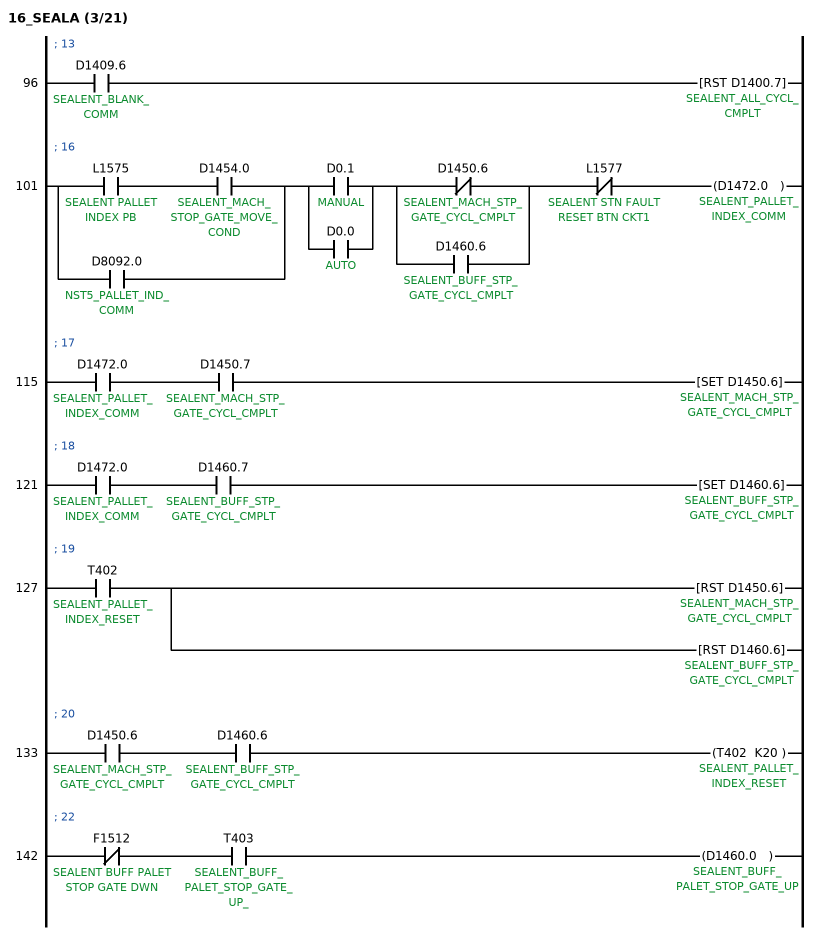
[picture p288: ladder of 16_SEALA, rungs at steps 96 to 142]
; 13
96    LD      D1409.6  ; SEALENT_BLANK_COMM
      RST     D1400.7  ; SEALENT_ALL_CYCL_CMPLT
; 16
101   LD      L1575  ; SEALENT PALLET INDEX PB
      AND     D1454.0  ; SEALENT_MACH_STOP_GATE_MOVE_COND
      OR      D8092.0  ; NST5_PALLET_IND_COMM
      LD      D0.1  ; MANUAL
      OR      D0.0  ; AUTO
      ANB
      LDI     D1450.6  ; SEALENT_MACH_STP_GATE_CYCL_CMPLT
      OR      D1460.6  ; SEALENT_BUFF_STP_GATE_CYCL_CMPLT
      ANB
      ANI     L1577  ; SEALENT STN FAULT RESET BTN CKT1
      OUT     D1472.0  ; SEALENT_PALLET_INDEX_COMM
; 17
115   LD      D1472.0  ; SEALENT_PALLET_INDEX_COMM
      AND     D1450.7  ; SEALENT_MACH_STP_GATE_CYCL_CMPLT
      SET     D1450.6  ; SEALENT_MACH_STP_GATE_CYCL_CMPLT
; 18
121   LD      D1472.0  ; SEALENT_PALLET_INDEX_COMM
      AND     D1460.7  ; SEALENT_BUFF_STP_GATE_CYCL_CMPLT
      SET     D1460.6  ; SEALENT_BUFF_STP_GATE_CYCL_CMPLT
; 19
127   LD      T402  ; SEALENT_PALLET_INDEX_RESET
      RST     D1450.6  ; SEALENT_MACH_STP_GATE_CYCL_CMPLT
      RST     D1460.6  ; SEALENT_BUFF_STP_GATE_CYCL_CMPLT
; 20
133   LD      D1450.6  ; SEALENT_MACH_STP_GATE_CYCL_CMPLT
      AND     D1460.6  ; SEALENT_BUFF_STP_GATE_CYCL_CMPLT
      OUT     T402 K20  ; SEALENT_PALLET_INDEX_RESET
; 22
142   LDI     F1512  ; SEALENT BUFF PALET STOP GATE DWN
      AND     T403  ; SEALENT_BUFF_PALET_STOP_GATE_UP_
      OUT     D1460.0  ; SEALENT_BUFF_PALET_STOP_GATE_UP
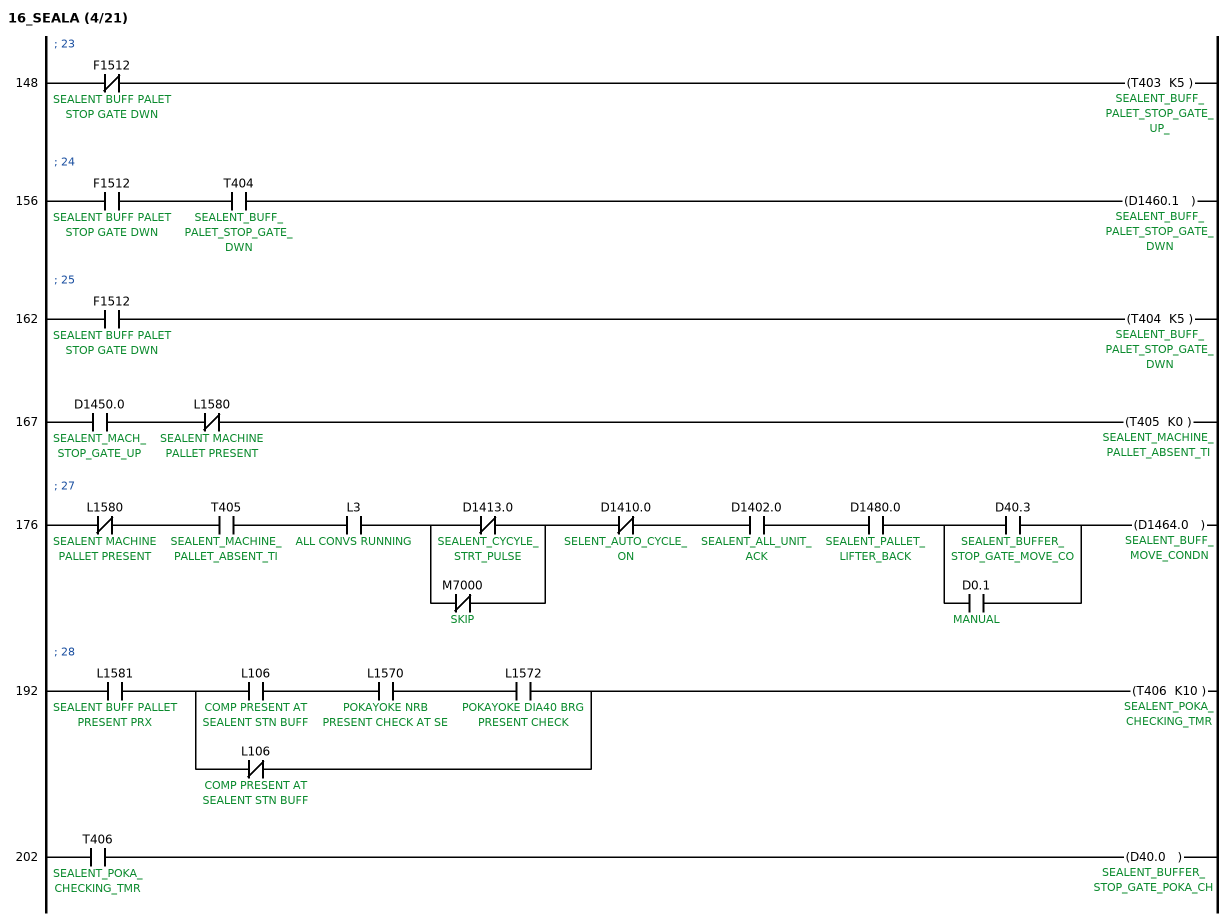
; 23
148   LDI     F1512  ; SEALENT BUFF PALET STOP GATE DWN
      OUT     T403 K5  ; SEALENT_BUFF_PALET_STOP_GATE_UP_
; 24
156   LD      F1512  ; SEALENT BUFF PALET STOP GATE DWN
      AND     T404  ; SEALENT_BUFF_PALET_STOP_GATE_DWN
      OUT     D1460.1  ; SEALENT_BUFF_PALET_STOP_GATE_DWN
; 25
162   LD      F1512  ; SEALENT BUFF PALET STOP GATE DWN
      OUT     T404 K5  ; SEALENT_BUFF_PALET_STOP_GATE_DWN
167   LD      D1450.0  ; SEALENT_MACH_STOP_GATE_UP
      ANI     L1580  ; SEALENT MACHINE PALLET PRESENT
      OUT     T405 K0  ; SEALENT_MACHINE_PALLET_ABSENT_TI
; 27
176   LDI     L1580  ; SEALENT MACHINE PALLET PRESENT
      AND     T405  ; SEALENT_MACHINE_PALLET_ABSENT_TI
      AND     L3  ; ALL CONVS RUNNING
      LDI     D1413.0  ; SEALENT_CYCYLE_STRT_PULSE
      ORI     M7000  ; SKIP
      ANB
      ANI     D1410.0  ; SELENT_AUTO_CYCLE_ON
      AND     D1402.0  ; SEALENT_ALL_UNIT_ACK
      AND     D1480.0  ; SEALENT_PALLET_LIFTER_BACK
      LD      D40.3  ; SEALENT_BUFFER_STOP_GATE_MOVE_CO
      OR      D0.1  ; MANUAL
      ANB
      OUT     D1464.0  ; SEALENT_BUFF_MOVE_CONDN
; 28
192   LD      L1581  ; SEALENT BUFF PALLET PRESENT PRX
      LD      L106  ; COMP PRESENT AT SEALENT STN BUFF
      AND     L1570  ; POKAYOKE NRB PRESENT CHECK AT SE
      AND     L1572  ; POKAYOKE DIA40 BRG PRESENT CHECK
      ORI     L106  ; COMP PRESENT AT SEALENT STN BUFF
      ANB
      OUT     T406 K10  ; SEALENT_POKA_CHECKING_TMR
202   LD      T406  ; SEALENT_POKA_CHECKING_TMR
      OUT     D40.0  ; SEALENT_BUFFER_STOP_GATE_POKA_CH
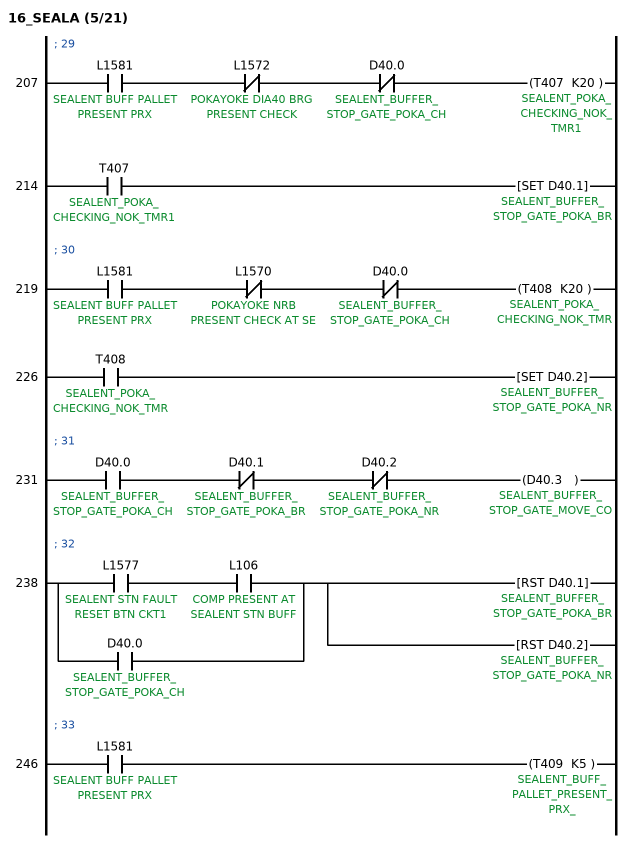
; 29
207   LD      L1581  ; SEALENT BUFF PALLET PRESENT PRX
      ANI     L1572  ; POKAYOKE DIA40 BRG PRESENT CHECK
      ANI     D40.0  ; SEALENT_BUFFER_STOP_GATE_POKA_CH
      OUT     T407 K20  ; SEALENT_POKA_CHECKING_NOK_TMR1
214   LD      T407  ; SEALENT_POKA_CHECKING_NOK_TMR1
      SET     D40.1  ; SEALENT_BUFFER_STOP_GATE_POKA_BR
; 30
219   LD      L1581  ; SEALENT BUFF PALLET PRESENT PRX
      ANI     L1570  ; POKAYOKE NRB PRESENT CHECK AT SE
      ANI     D40.0  ; SEALENT_BUFFER_STOP_GATE_POKA_CH
      OUT     T408 K20  ; SEALENT_POKA_CHECKING_NOK_TMR
226   LD      T408  ; SEALENT_POKA_CHECKING_NOK_TMR
      SET     D40.2  ; SEALENT_BUFFER_STOP_GATE_POKA_NR
; 31
231   LD      D40.0  ; SEALENT_BUFFER_STOP_GATE_POKA_CH
      ANI     D40.1  ; SEALENT_BUFFER_STOP_GATE_POKA_BR
      ANI     D40.2  ; SEALENT_BUFFER_STOP_GATE_POKA_NR
      OUT     D40.3  ; SEALENT_BUFFER_STOP_GATE_MOVE_CO
; 32
238   LD      L1577  ; SEALENT STN FAULT RESET BTN CKT1
      AND     L106  ; COMP PRESENT AT SEALENT STN BUFF
      OR      D40.0  ; SEALENT_BUFFER_STOP_GATE_POKA_CH
      RST     D40.1  ; SEALENT_BUFFER_STOP_GATE_POKA_BR
      RST     D40.2  ; SEALENT_BUFFER_STOP_GATE_POKA_NR
; 33
246   LD      L1581  ; SEALENT BUFF PALLET PRESENT PRX
      OUT     T409 K5  ; SEALENT_BUFF_PALLET_PRESENT_PRX_
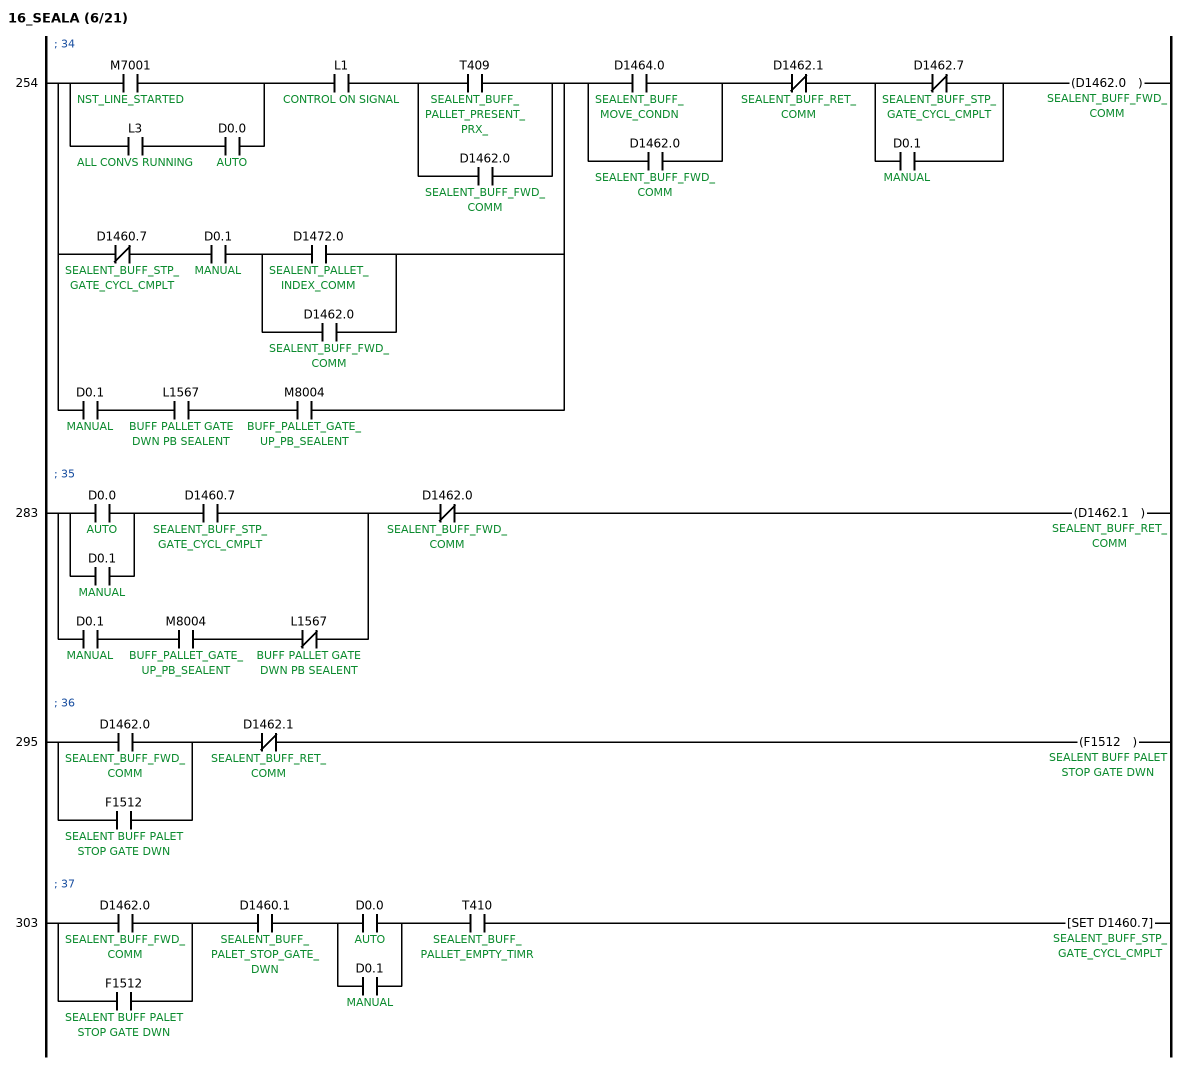
; 34
254   LD      M7001  ; NST_LINE_STARTED
      LD      L3  ; ALL CONVS RUNNING
      AND     D0.0  ; AUTO
      ORB
      AND     L1  ; CONTROL ON SIGNAL
      LD      T409  ; SEALENT_BUFF_PALLET_PRESENT_PRX_
      OR      D1462.0  ; SEALENT_BUFF_FWD_COMM
      ANB
      LDI     D1460.7  ; SEALENT_BUFF_STP_GATE_CYCL_CMPLT
      AND     D0.1  ; MANUAL
      LD      D1472.0  ; SEALENT_PALLET_INDEX_COMM
      OR      D1462.0  ; SEALENT_BUFF_FWD_COMM
      ANB
      ORB
      LD      D0.1  ; MANUAL
      AND     L1567  ; BUFF PALLET GATE DWN PB SEALENT
      AND     M8004  ; BUFF_PALLET_GATE_UP_PB_SEALENT
      ORB
      LD      D1464.0  ; SEALENT_BUFF_MOVE_CONDN
      OR      D1462.0  ; SEALENT_BUFF_FWD_COMM
      ANB
      ANI     D1462.1  ; SEALENT_BUFF_RET_COMM
      LDI     D1462.7  ; SEALENT_BUFF_STP_GATE_CYCL_CMPLT
      OR      D0.1  ; MANUAL
      ANB
      OUT     D1462.0  ; SEALENT_BUFF_FWD_COMM
; 35
283   LD      D0.0  ; AUTO
      OR      D0.1  ; MANUAL
      AND     D1460.7  ; SEALENT_BUFF_STP_GATE_CYCL_CMPLT
      LD      D0.1  ; MANUAL
      AND     M8004  ; BUFF_PALLET_GATE_UP_PB_SEALENT
      ANI     L1567  ; BUFF PALLET GATE DWN PB SEALENT
      ORB
      ANI     D1462.0  ; SEALENT_BUFF_FWD_COMM
      OUT     D1462.1  ; SEALENT_BUFF_RET_COMM
; 36
295   LD      D1462.0  ; SEALENT_BUFF_FWD_COMM
      OR      F1512  ; SEALENT BUFF PALET STOP GATE DWN
      ANI     D1462.1  ; SEALENT_BUFF_RET_COMM
      OUT     F1512  ; SEALENT BUFF PALET STOP GATE DWN
; 37
303   LD      D1462.0  ; SEALENT_BUFF_FWD_COMM
      OR      F1512  ; SEALENT BUFF PALET STOP GATE DWN
      AND     D1460.1  ; SEALENT_BUFF_PALET_STOP_GATE_DWN
      LD      D0.0  ; AUTO
      OR      D0.1  ; MANUAL
      ANB
      AND     T410  ; SEALENT_BUFF_PALLET_EMPTY_TIMR
      SET     D1460.7  ; SEALENT_BUFF_STP_GATE_CYCL_CMPLT
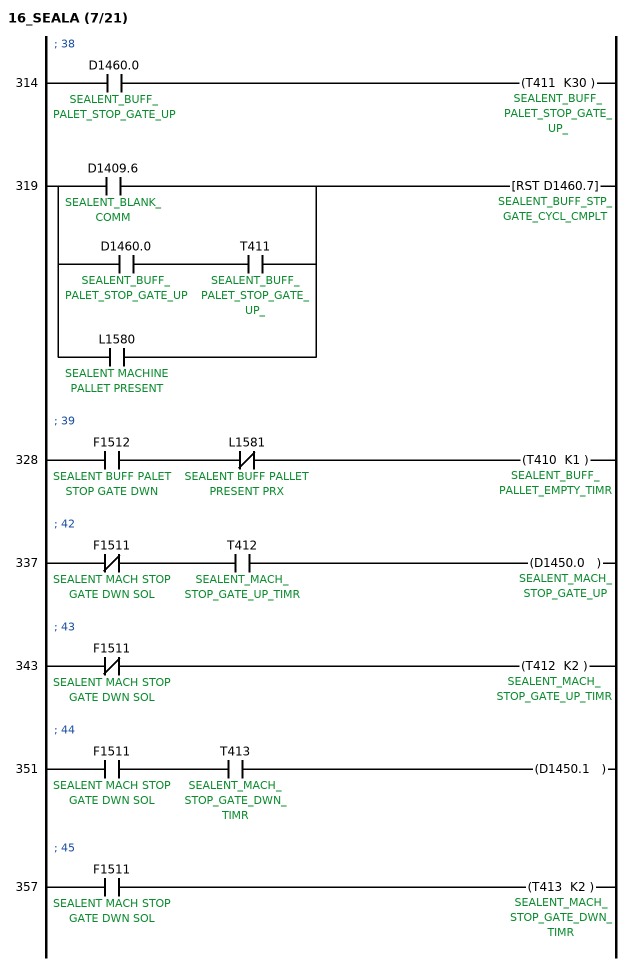
; 38
314   LD      D1460.0  ; SEALENT_BUFF_PALET_STOP_GATE_UP
      OUT     T411 K30  ; SEALENT_BUFF_PALET_STOP_GATE_UP_
319   LD      D1409.6  ; SEALENT_BLANK_COMM
      LD      D1460.0  ; SEALENT_BUFF_PALET_STOP_GATE_UP
      AND     T411  ; SEALENT_BUFF_PALET_STOP_GATE_UP_
      ORB
      OR      L1580  ; SEALENT MACHINE PALLET PRESENT
      RST     D1460.7  ; SEALENT_BUFF_STP_GATE_CYCL_CMPLT
; 39
328   LD      F1512  ; SEALENT BUFF PALET STOP GATE DWN
      ANI     L1581  ; SEALENT BUFF PALLET PRESENT PRX
      OUT     T410 K1  ; SEALENT_BUFF_PALLET_EMPTY_TIMR
; 42
337   LDI     F1511  ; SEALENT MACH STOP GATE DWN SOL
      AND     T412  ; SEALENT_MACH_STOP_GATE_UP_TIMR
      OUT     D1450.0  ; SEALENT_MACH_STOP_GATE_UP
; 43
343   LDI     F1511  ; SEALENT MACH STOP GATE DWN SOL
      OUT     T412 K2  ; SEALENT_MACH_STOP_GATE_UP_TIMR
; 44
351   LD      F1511  ; SEALENT MACH STOP GATE DWN SOL
      AND     T413  ; SEALENT_MACH_STOP_GATE_DWN_TIMR
      OUT     D1450.1
; 45
357   LD      F1511  ; SEALENT MACH STOP GATE DWN SOL
      OUT     T413 K2  ; SEALENT_MACH_STOP_GATE_DWN_TIMR
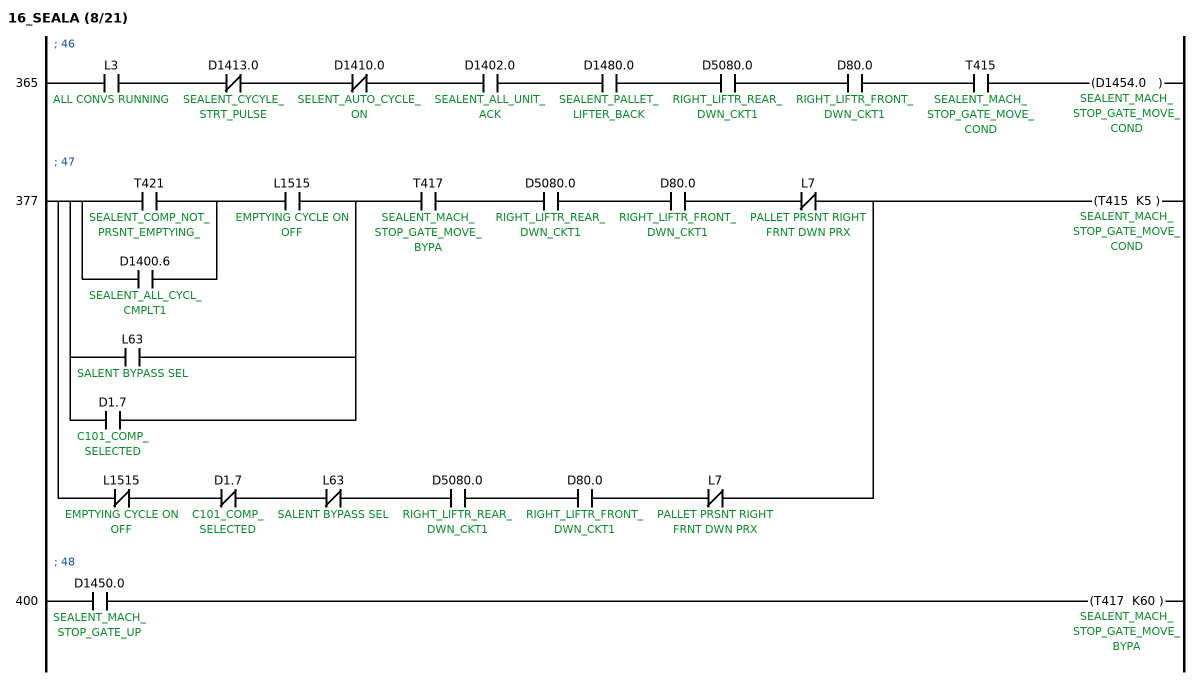
; 46
365   LD      L3  ; ALL CONVS RUNNING
      ANI     D1413.0  ; SEALENT_CYCYLE_STRT_PULSE
      ANI     D1410.0  ; SELENT_AUTO_CYCLE_ON
      AND     D1402.0  ; SEALENT_ALL_UNIT_ACK
      AND     D1480.0  ; SEALENT_PALLET_LIFTER_BACK
      AND     D5080.0  ; RIGHT_LIFTR_REAR_DWN_CKT1
      AND     D80.0  ; RIGHT_LIFTR_FRONT_DWN_CKT1
      AND     T415  ; SEALENT_MACH_STOP_GATE_MOVE_COND
      OUT     D1454.0  ; SEALENT_MACH_STOP_GATE_MOVE_COND
; 47
377   LD      T421  ; SEALENT_COMP_NOT_PRSNT_EMPTYING_
      OR      D1400.6  ; SEALENT_ALL_CYCL_CMPLT1
      AND     L1515  ; EMPTYING CYCLE ON OFF
      OR      L63  ; SALENT BYPASS SEL
      OR      D1.7  ; C101_COMP_SELECTED
      AND     T417  ; SEALENT_MACH_STOP_GATE_MOVE_BYPA
      AND     D5080.0  ; RIGHT_LIFTR_REAR_DWN_CKT1
      AND     D80.0  ; RIGHT_LIFTR_FRONT_DWN_CKT1
      ANI     L7  ; PALLET PRSNT RIGHT FRNT DWN PRX
      LDI     L1515  ; EMPTYING CYCLE ON OFF
      ANI     D1.7  ; C101_COMP_SELECTED
      ANI     L63  ; SALENT BYPASS SEL
      AND     D5080.0  ; RIGHT_LIFTR_REAR_DWN_CKT1
      AND     D80.0  ; RIGHT_LIFTR_FRONT_DWN_CKT1
      ANI     L7  ; PALLET PRSNT RIGHT FRNT DWN PRX
      ORB
      OUT     T415 K5  ; SEALENT_MACH_STOP_GATE_MOVE_COND
; 48
400   LD      D1450.0  ; SEALENT_MACH_STOP_GATE_UP
      OUT     T417 K60  ; SEALENT_MACH_STOP_GATE_MOVE_BYPA
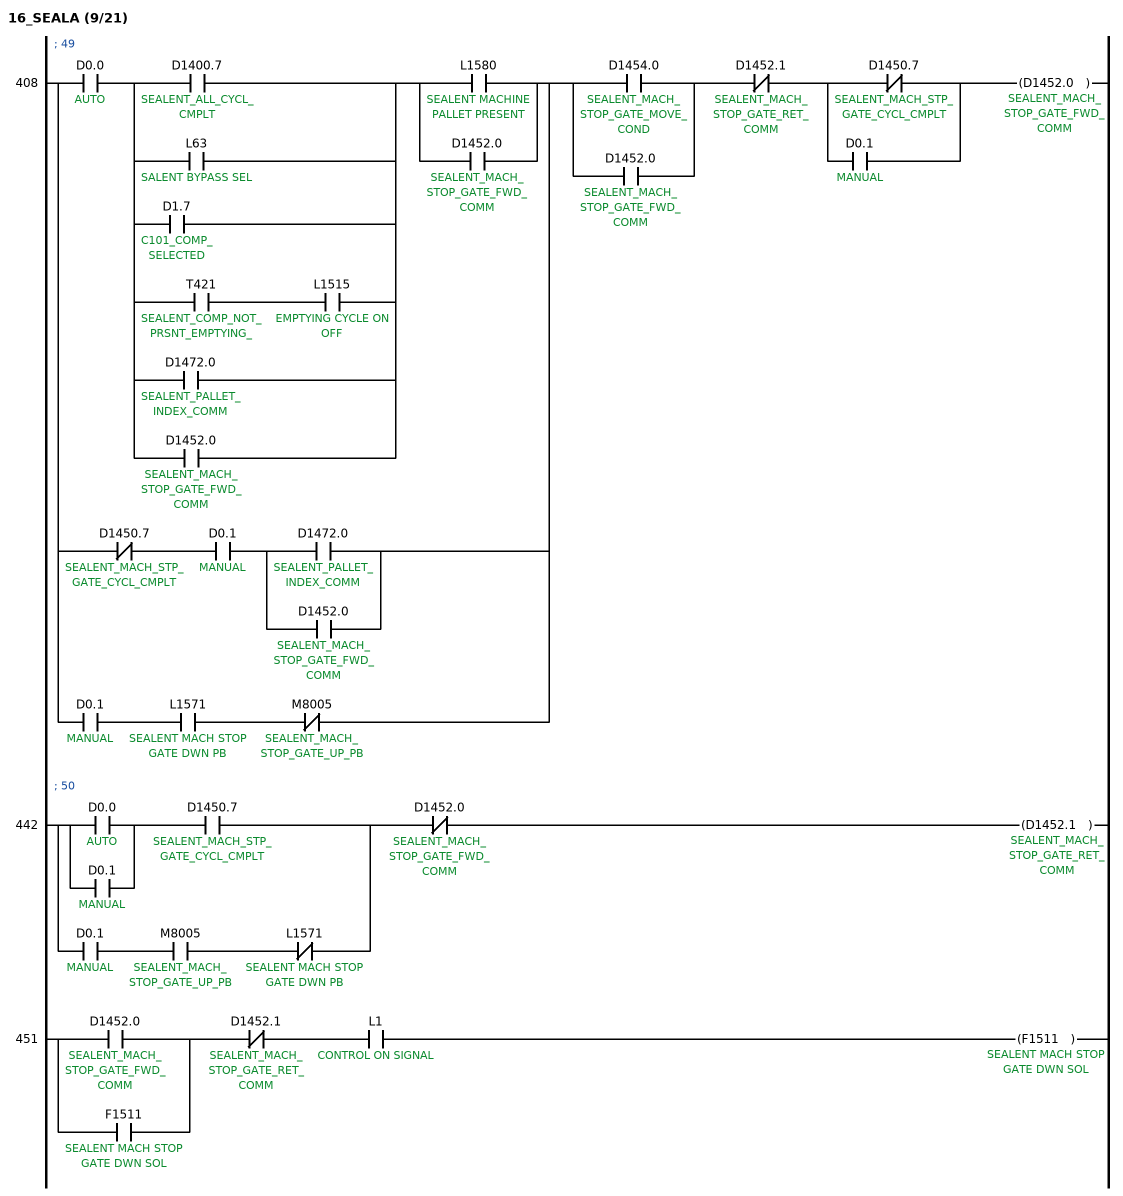
; 49
408   LD      D0.0  ; AUTO
      LD      D1400.7  ; SEALENT_ALL_CYCL_CMPLT
      OR      L63  ; SALENT BYPASS SEL
      OR      D1.7  ; C101_COMP_SELECTED
      LD      T421  ; SEALENT_COMP_NOT_PRSNT_EMPTYING_
      AND     L1515  ; EMPTYING CYCLE ON OFF
      ORB
      OR      D1472.0  ; SEALENT_PALLET_INDEX_COMM
      OR      D1452.0  ; SEALENT_MACH_STOP_GATE_FWD_COMM
      ANB
      LD      L1580  ; SEALENT MACHINE PALLET PRESENT
      OR      D1452.0  ; SEALENT_MACH_STOP_GATE_FWD_COMM
      ANB
      LDI     D1450.7  ; SEALENT_MACH_STP_GATE_CYCL_CMPLT
      AND     D0.1  ; MANUAL
      LD      D1472.0  ; SEALENT_PALLET_INDEX_COMM
      OR      D1452.0  ; SEALENT_MACH_STOP_GATE_FWD_COMM
      ANB
      ORB
      LD      D0.1  ; MANUAL
      AND     L1571  ; SEALENT MACH STOP GATE DWN PB
      ANI     M8005  ; SEALENT_MACH_STOP_GATE_UP_PB
      ORB
      LD      D1454.0  ; SEALENT_MACH_STOP_GATE_MOVE_COND
      OR      D1452.0  ; SEALENT_MACH_STOP_GATE_FWD_COMM
      ANB
      ANI     D1452.1  ; SEALENT_MACH_STOP_GATE_RET_COMM
      LDI     D1450.7  ; SEALENT_MACH_STP_GATE_CYCL_CMPLT
      OR      D0.1  ; MANUAL
      ANB
      OUT     D1452.0  ; SEALENT_MACH_STOP_GATE_FWD_COMM
; 50
442   LD      D0.0  ; AUTO
      OR      D0.1  ; MANUAL
      AND     D1450.7  ; SEALENT_MACH_STP_GATE_CYCL_CMPLT
      LD      D0.1  ; MANUAL
      AND     M8005  ; SEALENT_MACH_STOP_GATE_UP_PB
      ANI     L1571  ; SEALENT MACH STOP GATE DWN PB
      ORB
      ANI     D1452.0  ; SEALENT_MACH_STOP_GATE_FWD_COMM
      OUT     D1452.1  ; SEALENT_MACH_STOP_GATE_RET_COMM
451   LD      D1452.0  ; SEALENT_MACH_STOP_GATE_FWD_COMM
      OR      F1511  ; SEALENT MACH STOP GATE DWN SOL
      ANI     D1452.1  ; SEALENT_MACH_STOP_GATE_RET_COMM
      AND     L1  ; CONTROL ON SIGNAL
      OUT     F1511  ; SEALENT MACH STOP GATE DWN SOL
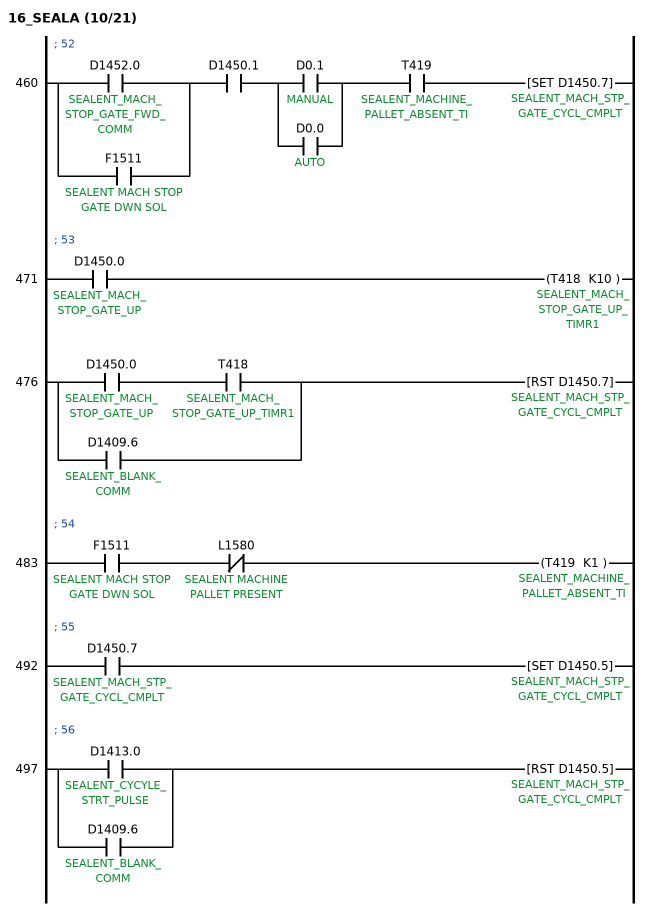
; 52
460   LD      D1452.0  ; SEALENT_MACH_STOP_GATE_FWD_COMM
      OR      F1511  ; SEALENT MACH STOP GATE DWN SOL
      AND     D1450.1
      LD      D0.1  ; MANUAL
      OR      D0.0  ; AUTO
      ANB
      AND     T419  ; SEALENT_MACHINE_PALLET_ABSENT_TI
      SET     D1450.7  ; SEALENT_MACH_STP_GATE_CYCL_CMPLT
; 53
471   LD      D1450.0  ; SEALENT_MACH_STOP_GATE_UP
      OUT     T418 K10  ; SEALENT_MACH_STOP_GATE_UP_TIMR1
476   LD      D1450.0  ; SEALENT_MACH_STOP_GATE_UP
      AND     T418  ; SEALENT_MACH_STOP_GATE_UP_TIMR1
      OR      D1409.6  ; SEALENT_BLANK_COMM
      RST     D1450.7  ; SEALENT_MACH_STP_GATE_CYCL_CMPLT
; 54
483   LD      F1511  ; SEALENT MACH STOP GATE DWN SOL
      ANI     L1580  ; SEALENT MACHINE PALLET PRESENT
      OUT     T419 K1  ; SEALENT_MACHINE_PALLET_ABSENT_TI
; 55
492   LD      D1450.7  ; SEALENT_MACH_STP_GATE_CYCL_CMPLT
      SET     D1450.5  ; SEALENT_MACH_STP_GATE_CYCL_CMPLT
; 56
497   LD      D1413.0  ; SEALENT_CYCYLE_STRT_PULSE
      OR      D1409.6  ; SEALENT_BLANK_COMM
      RST     D1450.5  ; SEALENT_MACH_STP_GATE_CYCL_CMPLT
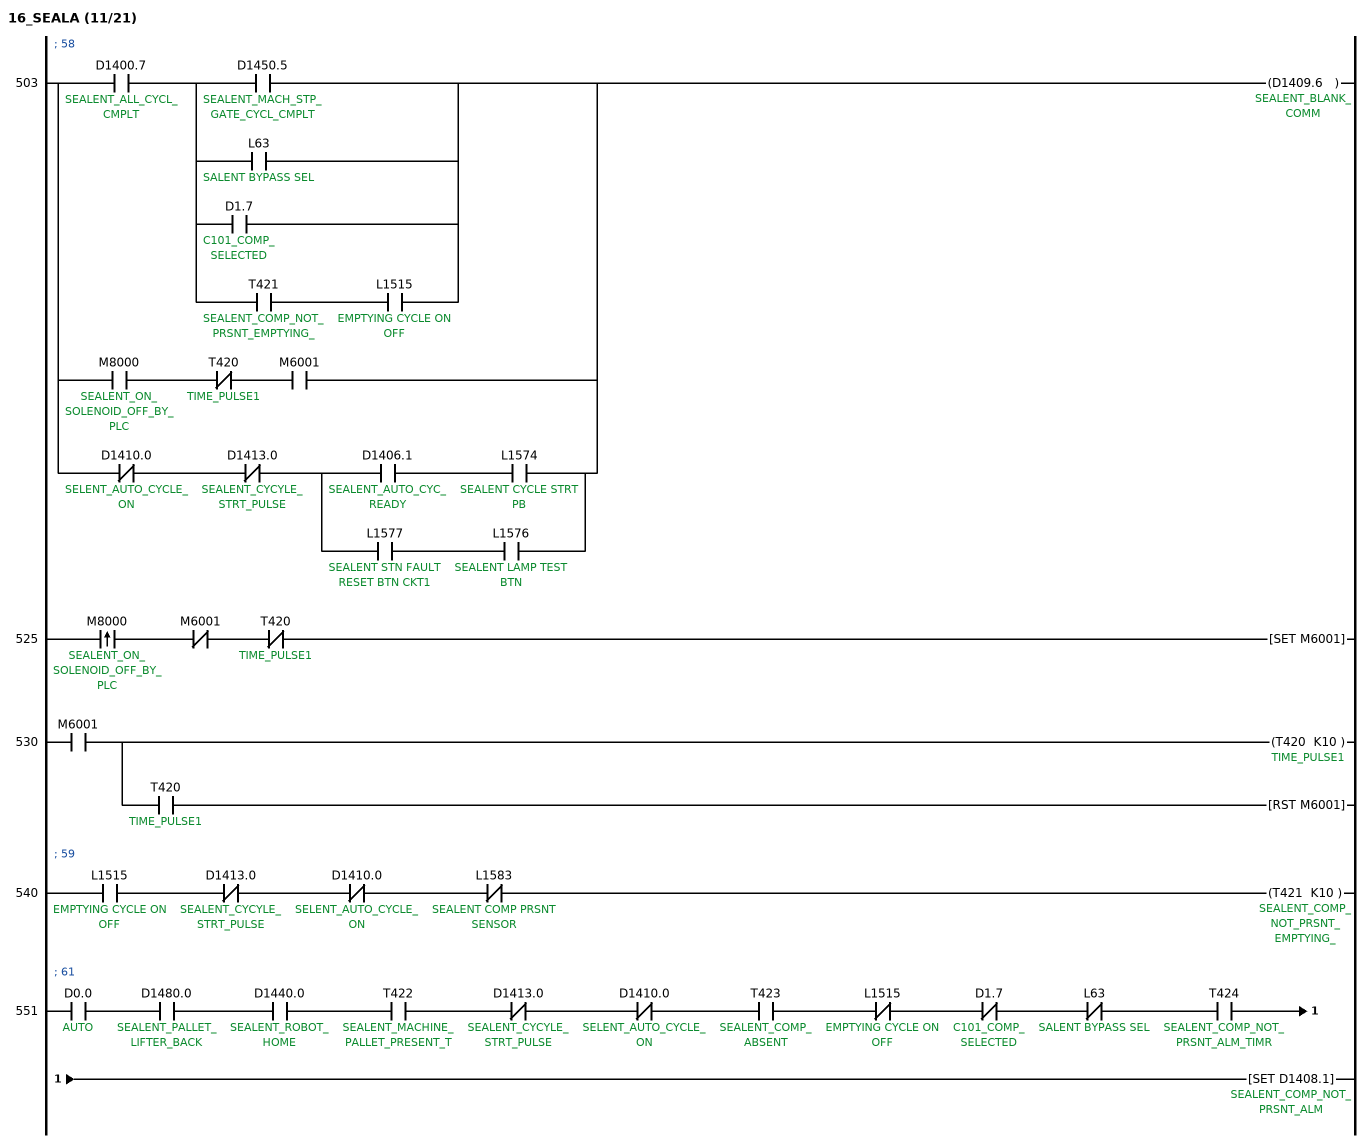
; 58
503   LD      D1400.7  ; SEALENT_ALL_CYCL_CMPLT
      LD      D1450.5  ; SEALENT_MACH_STP_GATE_CYCL_CMPLT
      OR      L63  ; SALENT BYPASS SEL
      OR      D1.7  ; C101_COMP_SELECTED
      LD      T421  ; SEALENT_COMP_NOT_PRSNT_EMPTYING_
      AND     L1515  ; EMPTYING CYCLE ON OFF
      ORB
      ANB
      LD      M8000  ; SEALENT_ON_SOLENOID_OFF_BY_PLC
      ANI     T420  ; TIME_PULSE1
      AND     M6001
      ORB
      LDI     D1410.0  ; SELENT_AUTO_CYCLE_ON
      ANI     D1413.0  ; SEALENT_CYCYLE_STRT_PULSE
      LD      D1406.1  ; SEALENT_AUTO_CYC_READY
      AND     L1574  ; SEALENT CYCLE STRT PB
      LD      L1577  ; SEALENT STN FAULT RESET BTN CKT1
      AND     L1576  ; SEALENT LAMP TEST BTN
      ORB
      ANB
      ORB
      OUT     D1409.6  ; SEALENT_BLANK_COMM
525   LDP     M8000  ; SEALENT_ON_SOLENOID_OFF_BY_PLC
      ANI     M6001
      ANI     T420  ; TIME_PULSE1
      SET     M6001
530   LD      M6001
      OUT     T420 K10  ; TIME_PULSE1
      AND     T420  ; TIME_PULSE1
      RST     M6001
; 59
540   LD      L1515  ; EMPTYING CYCLE ON OFF
      ANI     D1413.0  ; SEALENT_CYCYLE_STRT_PULSE
      ANI     D1410.0  ; SELENT_AUTO_CYCLE_ON
      ANI     L1583  ; SEALENT COMP PRSNT SENSOR
      OUT     T421 K10  ; SEALENT_COMP_NOT_PRSNT_EMPTYING_
; 61
551   LD      D0.0  ; AUTO
      AND     D1480.0  ; SEALENT_PALLET_LIFTER_BACK
      AND     D1440.0  ; SEALENT_ROBOT_HOME
      AND     T422  ; SEALENT_MACHINE_PALLET_PRESENT_T
      ANI     D1413.0  ; SEALENT_CYCYLE_STRT_PULSE
      ANI     D1410.0  ; SELENT_AUTO_CYCLE_ON
      AND     T423  ; SEALENT_COMP_ABSENT
      ANI     L1515  ; EMPTYING CYCLE ON OFF
      ANI     D1.7  ; C101_COMP_SELECTED
      ANI     L63  ; SALENT BYPASS SEL
      AND     T424  ; SEALENT_COMP_NOT_PRSNT_ALM_TIMR
      SET     D1408.1  ; SEALENT_COMP_NOT_PRSNT_ALM
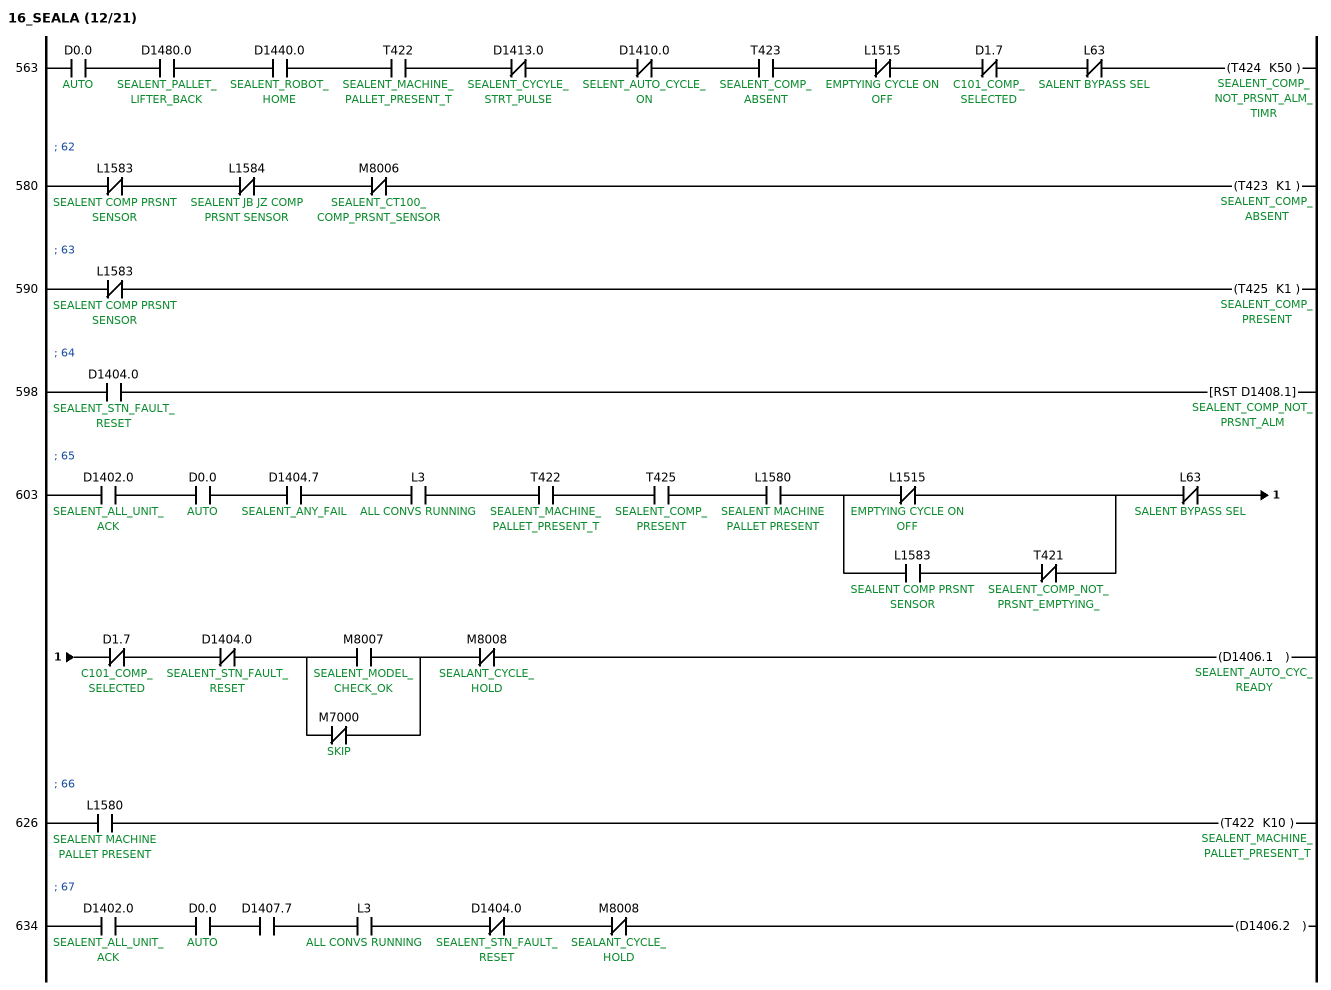
563   LD      D0.0  ; AUTO
      AND     D1480.0  ; SEALENT_PALLET_LIFTER_BACK
      AND     D1440.0  ; SEALENT_ROBOT_HOME
      AND     T422  ; SEALENT_MACHINE_PALLET_PRESENT_T
      ANI     D1413.0  ; SEALENT_CYCYLE_STRT_PULSE
      ANI     D1410.0  ; SELENT_AUTO_CYCLE_ON
      AND     T423  ; SEALENT_COMP_ABSENT
      ANI     L1515  ; EMPTYING CYCLE ON OFF
      ANI     D1.7  ; C101_COMP_SELECTED
      ANI     L63  ; SALENT BYPASS SEL
      OUT     T424 K50  ; SEALENT_COMP_NOT_PRSNT_ALM_TIMR
; 62
580   LDI     L1583  ; SEALENT COMP PRSNT SENSOR
      ANI     L1584  ; SEALENT JB JZ COMP PRSNT SENSOR
      ANI     M8006  ; SEALENT_CT100_COMP_PRSNT_SENSOR
      OUT     T423 K1  ; SEALENT_COMP_ABSENT
; 63
590   LDI     L1583  ; SEALENT COMP PRSNT SENSOR
      OUT     T425 K1  ; SEALENT_COMP_PRESENT
; 64
598   LD      D1404.0  ; SEALENT_STN_FAULT_RESET
      RST     D1408.1  ; SEALENT_COMP_NOT_PRSNT_ALM
; 65
603   LD      D1402.0  ; SEALENT_ALL_UNIT_ACK
      AND     D0.0  ; AUTO
      AND     D1404.7  ; SEALENT_ANY_FAIL
      AND     L3  ; ALL CONVS RUNNING
      AND     T422  ; SEALENT_MACHINE_PALLET_PRESENT_T
      AND     T425  ; SEALENT_COMP_PRESENT
      AND     L1580  ; SEALENT MACHINE PALLET PRESENT
      LDI     L1515  ; EMPTYING CYCLE ON OFF
      LD      L1583  ; SEALENT COMP PRSNT SENSOR
      ANI     T421  ; SEALENT_COMP_NOT_PRSNT_EMPTYING_
      ORB
      ANB
      ANI     L63  ; SALENT BYPASS SEL
      ANI     D1.7  ; C101_COMP_SELECTED
      ANI     D1404.0  ; SEALENT_STN_FAULT_RESET
      LD      M8007  ; SEALENT_MODEL_CHECK_OK
      ORI     M7000  ; SKIP
      ANB
      ANI     M8008  ; SEALANT_CYCLE_HOLD
      OUT     D1406.1  ; SEALENT_AUTO_CYC_READY
; 66
626   LD      L1580  ; SEALENT MACHINE PALLET PRESENT
      OUT     T422 K10  ; SEALENT_MACHINE_PALLET_PRESENT_T
; 67
634   LD      D1402.0  ; SEALENT_ALL_UNIT_ACK
      AND     D0.0  ; AUTO
      AND     D1407.7
      AND     L3  ; ALL CONVS RUNNING
      ANI     D1404.0  ; SEALENT_STN_FAULT_RESET
      ANI     M8008  ; SEALANT_CYCLE_HOLD
      OUT     D1406.2
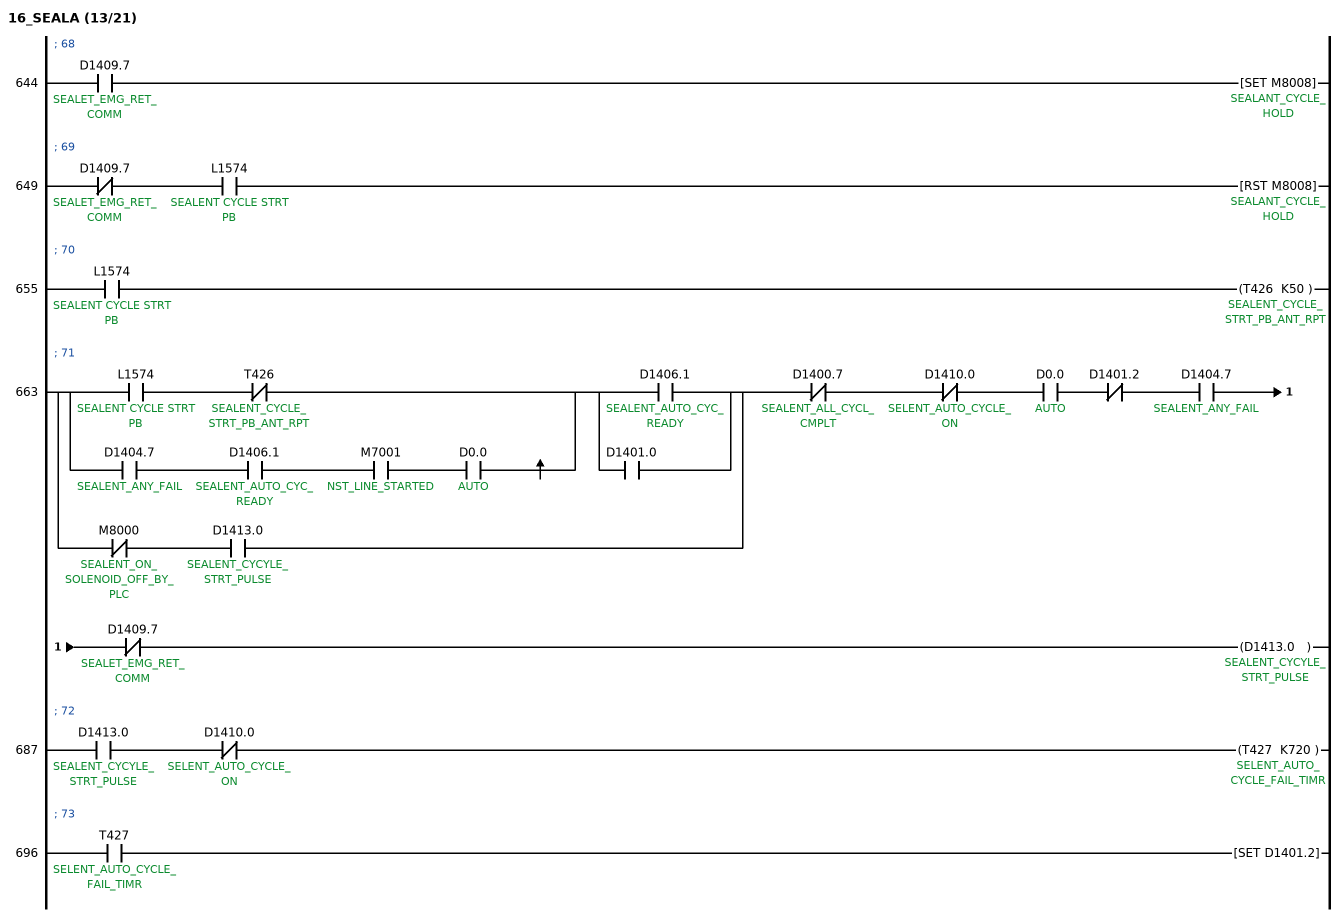
; 68
644   LD      D1409.7  ; SEALET_EMG_RET_COMM
      SET     M8008  ; SEALANT_CYCLE_HOLD
; 69
649   LDI     D1409.7  ; SEALET_EMG_RET_COMM
      AND     L1574  ; SEALENT CYCLE STRT PB
      RST     M8008  ; SEALANT_CYCLE_HOLD
; 70
655   LD      L1574  ; SEALENT CYCLE STRT PB
      OUT     T426 K50  ; SEALENT_CYCLE_STRT_PB_ANT_RPT
; 71
663   LD      L1574  ; SEALENT CYCLE STRT PB
      ANI     T426  ; SEALENT_CYCLE_STRT_PB_ANT_RPT
      LD      D1404.7  ; SEALENT_ANY_FAIL
      AND     D1406.1  ; SEALENT_AUTO_CYC_READY
      AND     M7001  ; NST_LINE_STARTED
      AND     D0.0  ; AUTO
      MEP
      ORB
      LD      D1406.1  ; SEALENT_AUTO_CYC_READY
      OR      D1401.0
      ANB
      LDI     M8000  ; SEALENT_ON_SOLENOID_OFF_BY_PLC
      AND     D1413.0  ; SEALENT_CYCYLE_STRT_PULSE
      ORB
      ANI     D1400.7  ; SEALENT_ALL_CYCL_CMPLT
      ANI     D1410.0  ; SELENT_AUTO_CYCLE_ON
      AND     D0.0  ; AUTO
      ANI     D1401.2
      AND     D1404.7  ; SEALENT_ANY_FAIL
      ANI     D1409.7  ; SEALET_EMG_RET_COMM
      OUT     D1413.0  ; SEALENT_CYCYLE_STRT_PULSE
; 72
687   LD      D1413.0  ; SEALENT_CYCYLE_STRT_PULSE
      ANI     D1410.0  ; SELENT_AUTO_CYCLE_ON
      OUT     T427 K720  ; SELENT_AUTO_CYCLE_FAIL_TIMR
; 73
696   LD      T427  ; SELENT_AUTO_CYCLE_FAIL_TIMR
      SET     D1401.2
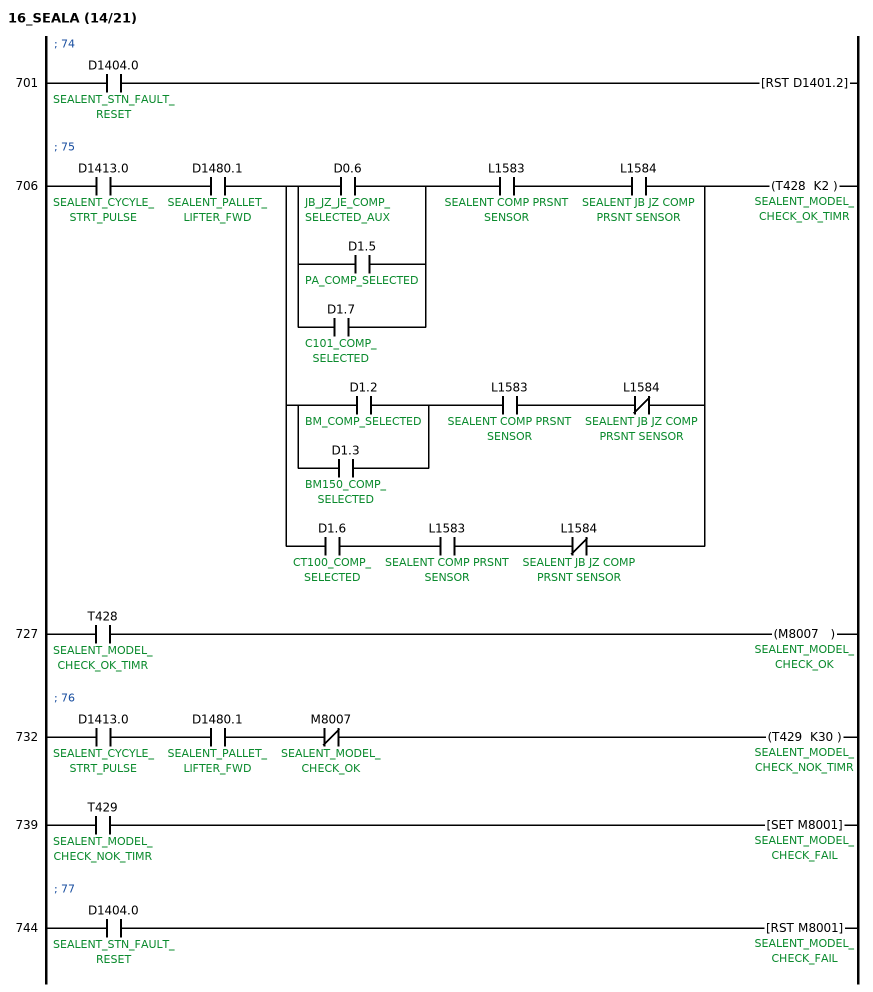
; 74
701   LD      D1404.0  ; SEALENT_STN_FAULT_RESET
      RST     D1401.2
; 75
706   LD      D1413.0  ; SEALENT_CYCYLE_STRT_PULSE
      AND     D1480.1  ; SEALENT_PALLET_LIFTER_FWD
      LD      D0.6  ; JB_JZ_JE_COMP_SELECTED_AUX
      OR      D1.5  ; PA_COMP_SELECTED
      OR      D1.7  ; C101_COMP_SELECTED
      AND     L1583  ; SEALENT COMP PRSNT SENSOR
      AND     L1584  ; SEALENT JB JZ COMP PRSNT SENSOR
      LD      D1.2  ; BM_COMP_SELECTED
      OR      D1.3  ; BM150_COMP_SELECTED
      AND     L1583  ; SEALENT COMP PRSNT SENSOR
      ANI     L1584  ; SEALENT JB JZ COMP PRSNT SENSOR
      ORB
      LD      D1.6  ; CT100_COMP_SELECTED
      AND     L1583  ; SEALENT COMP PRSNT SENSOR
      ANI     L1584  ; SEALENT JB JZ COMP PRSNT SENSOR
      ORB
      ANB
      OUT     T428 K2  ; SEALENT_MODEL_CHECK_OK_TIMR
727   LD      T428  ; SEALENT_MODEL_CHECK_OK_TIMR
      OUT     M8007  ; SEALENT_MODEL_CHECK_OK
; 76
732   LD      D1413.0  ; SEALENT_CYCYLE_STRT_PULSE
      AND     D1480.1  ; SEALENT_PALLET_LIFTER_FWD
      ANI     M8007  ; SEALENT_MODEL_CHECK_OK
      OUT     T429 K30  ; SEALENT_MODEL_CHECK_NOK_TIMR
739   LD      T429  ; SEALENT_MODEL_CHECK_NOK_TIMR
      SET     M8001  ; SEALENT_MODEL_CHECK_FAIL
; 77
744   LD      D1404.0  ; SEALENT_STN_FAULT_RESET
      RST     M8001  ; SEALENT_MODEL_CHECK_FAIL
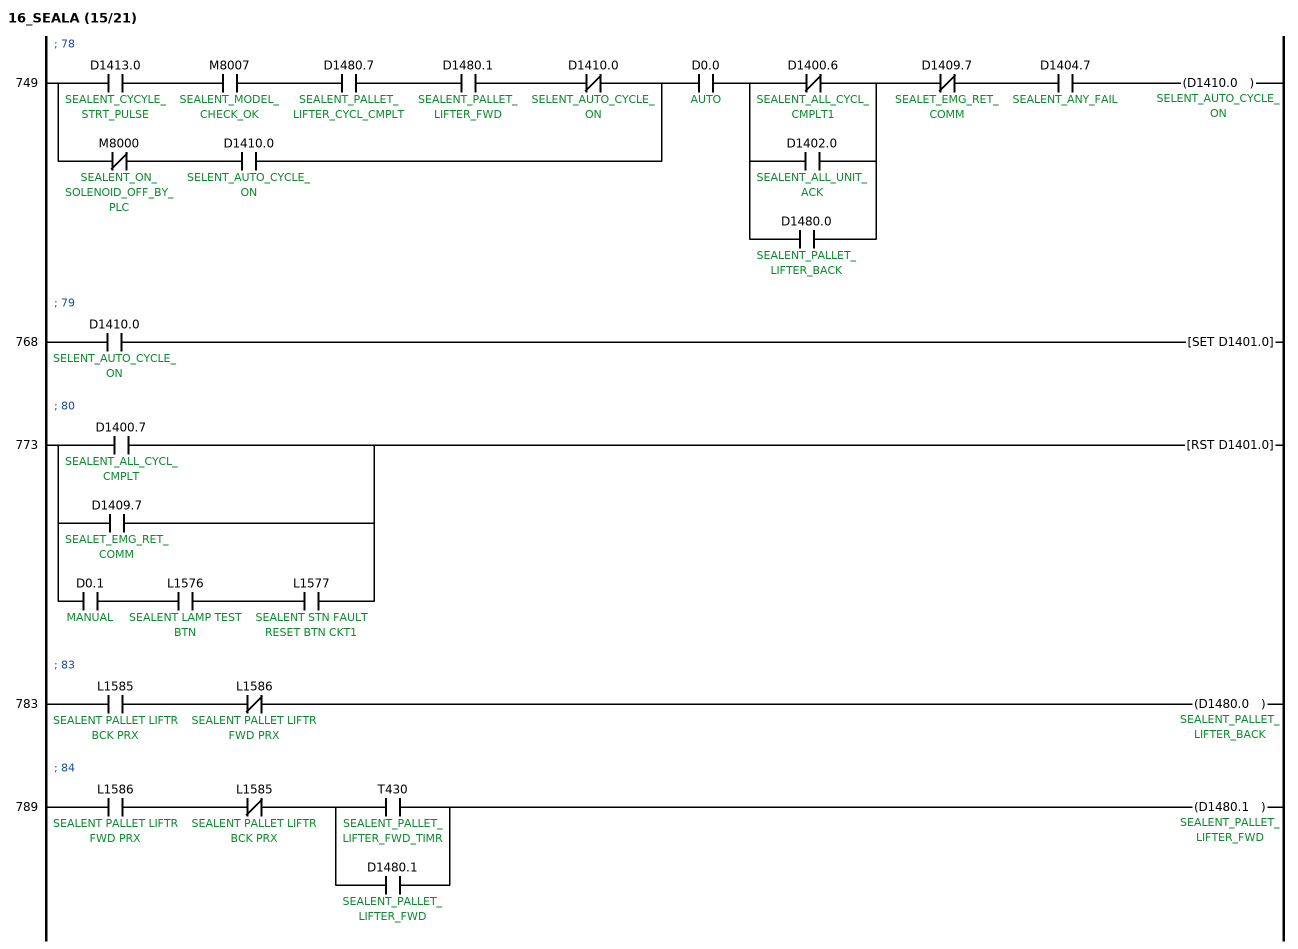
; 78
749   LD      D1413.0  ; SEALENT_CYCYLE_STRT_PULSE
      AND     M8007  ; SEALENT_MODEL_CHECK_OK
      AND     D1480.7  ; SEALENT_PALLET_LIFTER_CYCL_CMPLT
      AND     D1480.1  ; SEALENT_PALLET_LIFTER_FWD
      ANI     D1410.0  ; SELENT_AUTO_CYCLE_ON
      LDI     M8000  ; SEALENT_ON_SOLENOID_OFF_BY_PLC
      AND     D1410.0  ; SELENT_AUTO_CYCLE_ON
      ORB
      AND     D0.0  ; AUTO
      LDI     D1400.6  ; SEALENT_ALL_CYCL_CMPLT1
      OR      D1402.0  ; SEALENT_ALL_UNIT_ACK
      OR      D1480.0  ; SEALENT_PALLET_LIFTER_BACK
      ANB
      ANI     D1409.7  ; SEALET_EMG_RET_COMM
      AND     D1404.7  ; SEALENT_ANY_FAIL
      OUT     D1410.0  ; SELENT_AUTO_CYCLE_ON
; 79
768   LD      D1410.0  ; SELENT_AUTO_CYCLE_ON
      SET     D1401.0
; 80
773   LD      D1400.7  ; SEALENT_ALL_CYCL_CMPLT
      OR      D1409.7  ; SEALET_EMG_RET_COMM
      LD      D0.1  ; MANUAL
      AND     L1576  ; SEALENT LAMP TEST BTN
      AND     L1577  ; SEALENT STN FAULT RESET BTN CKT1
      ORB
      RST     D1401.0
; 83
783   LD      L1585  ; SEALENT PALLET LIFTR BCK PRX
      ANI     L1586  ; SEALENT PALLET LIFTR FWD PRX
      OUT     D1480.0  ; SEALENT_PALLET_LIFTER_BACK
; 84
789   LD      L1586  ; SEALENT PALLET LIFTR FWD PRX
      ANI     L1585  ; SEALENT PALLET LIFTR BCK PRX
      LD      T430  ; SEALENT_PALLET_LIFTER_FWD_TIMR
      OR      D1480.1  ; SEALENT_PALLET_LIFTER_FWD
      ANB
      OUT     D1480.1  ; SEALENT_PALLET_LIFTER_FWD
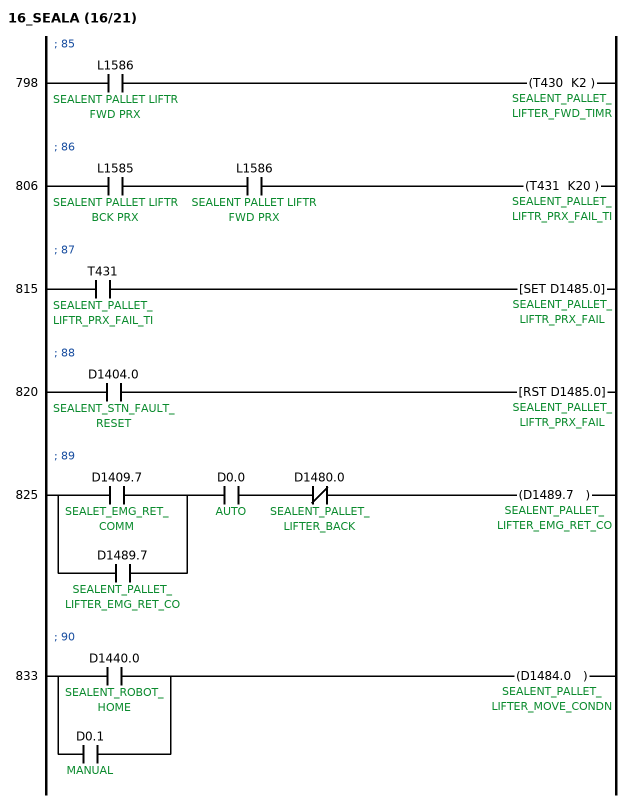
; 85
798   LD      L1586  ; SEALENT PALLET LIFTR FWD PRX
      OUT     T430 K2  ; SEALENT_PALLET_LIFTER_FWD_TIMR
; 86
806   LD      L1585  ; SEALENT PALLET LIFTR BCK PRX
      AND     L1586  ; SEALENT PALLET LIFTR FWD PRX
      OUT     T431 K20  ; SEALENT_PALLET_LIFTR_PRX_FAIL_TI
; 87
815   LD      T431  ; SEALENT_PALLET_LIFTR_PRX_FAIL_TI
      SET     D1485.0  ; SEALENT_PALLET_LIFTR_PRX_FAIL
; 88
820   LD      D1404.0  ; SEALENT_STN_FAULT_RESET
      RST     D1485.0  ; SEALENT_PALLET_LIFTR_PRX_FAIL
; 89
825   LD      D1409.7  ; SEALET_EMG_RET_COMM
      OR      D1489.7  ; SEALENT_PALLET_LIFTER_EMG_RET_CO
      AND     D0.0  ; AUTO
      ANI     D1480.0  ; SEALENT_PALLET_LIFTER_BACK
      OUT     D1489.7  ; SEALENT_PALLET_LIFTER_EMG_RET_CO
; 90
833   LD      D1440.0  ; SEALENT_ROBOT_HOME
      OR      D0.1  ; MANUAL
      OUT     D1484.0  ; SEALENT_PALLET_LIFTER_MOVE_CONDN
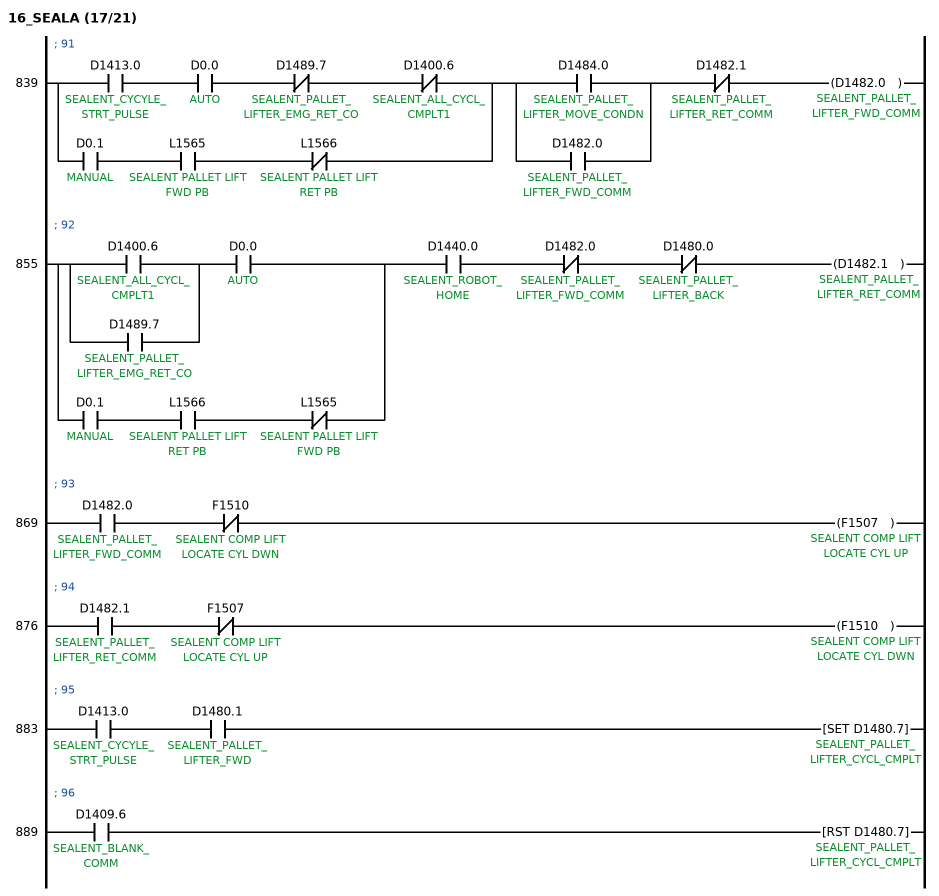
; 91
839   LD      D1413.0  ; SEALENT_CYCYLE_STRT_PULSE
      AND     D0.0  ; AUTO
      ANI     D1489.7  ; SEALENT_PALLET_LIFTER_EMG_RET_CO
      ANI     D1400.6  ; SEALENT_ALL_CYCL_CMPLT1
      LD      D0.1  ; MANUAL
      AND     L1565  ; SEALENT PALLET LIFT FWD PB
      ANI     L1566  ; SEALENT PALLET LIFT RET PB
      ORB
      LD      D1484.0  ; SEALENT_PALLET_LIFTER_MOVE_CONDN
      OR      D1482.0  ; SEALENT_PALLET_LIFTER_FWD_COMM
      ANB
      ANI     D1482.1  ; SEALENT_PALLET_LIFTER_RET_COMM
      OUT     D1482.0  ; SEALENT_PALLET_LIFTER_FWD_COMM
; 92
855   LD      D1400.6  ; SEALENT_ALL_CYCL_CMPLT1
      OR      D1489.7  ; SEALENT_PALLET_LIFTER_EMG_RET_CO
      AND     D0.0  ; AUTO
      LD      D0.1  ; MANUAL
      AND     L1566  ; SEALENT PALLET LIFT RET PB
      ANI     L1565  ; SEALENT PALLET LIFT FWD PB
      ORB
      AND     D1440.0  ; SEALENT_ROBOT_HOME
      ANI     D1482.0  ; SEALENT_PALLET_LIFTER_FWD_COMM
      ANI     D1480.0  ; SEALENT_PALLET_LIFTER_BACK
      OUT     D1482.1  ; SEALENT_PALLET_LIFTER_RET_COMM
; 93
869   LD      D1482.0  ; SEALENT_PALLET_LIFTER_FWD_COMM
      ANI     F1510  ; SEALENT COMP LIFT LOCATE CYL DWN
      OUT     F1507  ; SEALENT COMP LIFT LOCATE CYL UP
; 94
876   LD      D1482.1  ; SEALENT_PALLET_LIFTER_RET_COMM
      ANI     F1507  ; SEALENT COMP LIFT LOCATE CYL UP
      OUT     F1510  ; SEALENT COMP LIFT LOCATE CYL DWN
; 95
883   LD      D1413.0  ; SEALENT_CYCYLE_STRT_PULSE
      AND     D1480.1  ; SEALENT_PALLET_LIFTER_FWD
      SET     D1480.7  ; SEALENT_PALLET_LIFTER_CYCL_CMPLT
; 96
889   LD      D1409.6  ; SEALENT_BLANK_COMM
      RST     D1480.7  ; SEALENT_PALLET_LIFTER_CYCL_CMPLT
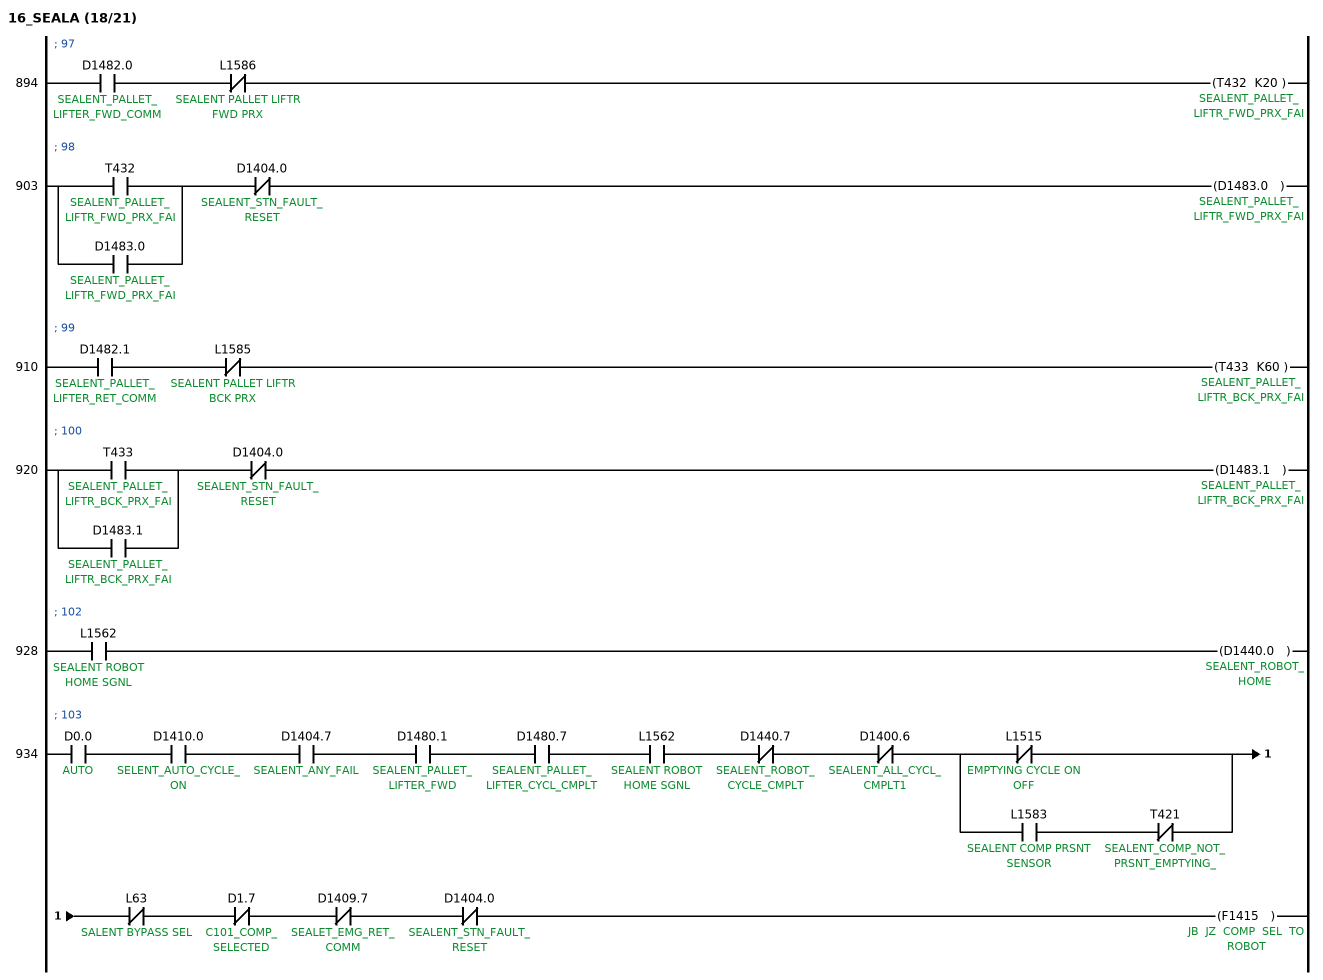
; 97
894   LD      D1482.0  ; SEALENT_PALLET_LIFTER_FWD_COMM
      ANI     L1586  ; SEALENT PALLET LIFTR FWD PRX
      OUT     T432 K20  ; SEALENT_PALLET_LIFTR_FWD_PRX_FAI
; 98
903   LD      T432  ; SEALENT_PALLET_LIFTR_FWD_PRX_FAI
      OR      D1483.0  ; SEALENT_PALLET_LIFTR_FWD_PRX_FAI
      ANI     D1404.0  ; SEALENT_STN_FAULT_RESET
      OUT     D1483.0  ; SEALENT_PALLET_LIFTR_FWD_PRX_FAI
; 99
910   LD      D1482.1  ; SEALENT_PALLET_LIFTER_RET_COMM
      ANI     L1585  ; SEALENT PALLET LIFTR BCK PRX
      OUT     T433 K60  ; SEALENT_PALLET_LIFTR_BCK_PRX_FAI
; 100
920   LD      T433  ; SEALENT_PALLET_LIFTR_BCK_PRX_FAI
      OR      D1483.1  ; SEALENT_PALLET_LIFTR_BCK_PRX_FAI
      ANI     D1404.0  ; SEALENT_STN_FAULT_RESET
      OUT     D1483.1  ; SEALENT_PALLET_LIFTR_BCK_PRX_FAI
; 102
928   LD      L1562  ; SEALENT ROBOT HOME SGNL
      OUT     D1440.0  ; SEALENT_ROBOT_HOME
; 103
934   LD      D0.0  ; AUTO
      AND     D1410.0  ; SELENT_AUTO_CYCLE_ON
      AND     D1404.7  ; SEALENT_ANY_FAIL
      AND     D1480.1  ; SEALENT_PALLET_LIFTER_FWD
      AND     D1480.7  ; SEALENT_PALLET_LIFTER_CYCL_CMPLT
      AND     L1562  ; SEALENT ROBOT HOME SGNL
      ANI     D1440.7  ; SEALENT_ROBOT_CYCLE_CMPLT
      ANI     D1400.6  ; SEALENT_ALL_CYCL_CMPLT1
      LDI     L1515  ; EMPTYING CYCLE ON OFF
      LD      L1583  ; SEALENT COMP PRSNT SENSOR
      ANI     T421  ; SEALENT_COMP_NOT_PRSNT_EMPTYING_
      ORB
      ANB
      ANI     L63  ; SALENT BYPASS SEL
      ANI     D1.7  ; C101_COMP_SELECTED
      ANI     D1409.7  ; SEALET_EMG_RET_COMM
      ANI     D1404.0  ; SEALENT_STN_FAULT_RESET
      OUT     F1415  ; JB  JZ  COMP  SEL  TO  ROBOT
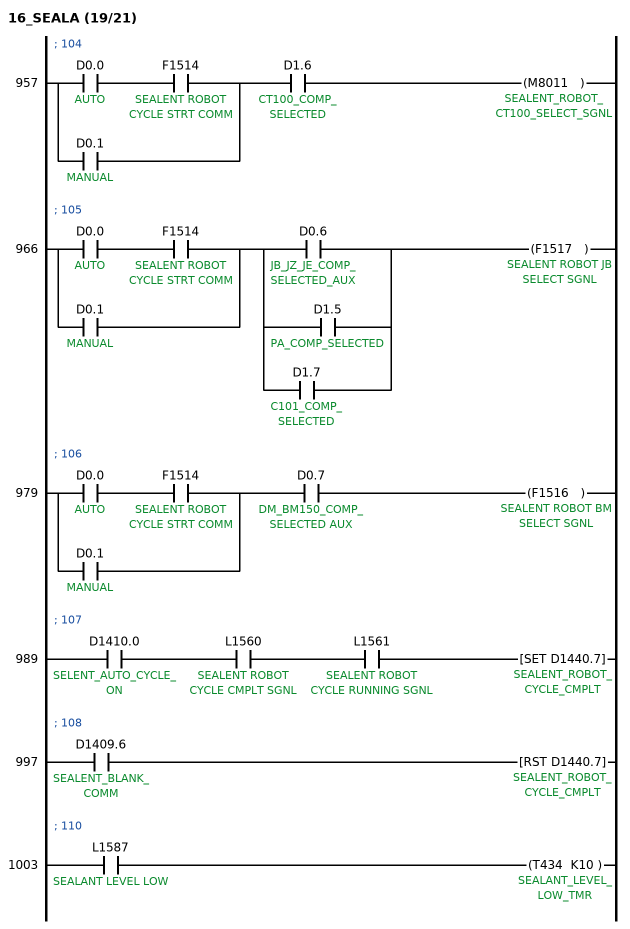
; 104
957   LD      D0.0  ; AUTO
      AND     F1514  ; SEALENT ROBOT CYCLE STRT COMM
      OR      D0.1  ; MANUAL
      AND     D1.6  ; CT100_COMP_SELECTED
      OUT     M8011  ; SEALENT_ROBOT_CT100_SELECT_SGNL
; 105
966   LD      D0.0  ; AUTO
      AND     F1514  ; SEALENT ROBOT CYCLE STRT COMM
      OR      D0.1  ; MANUAL
      LD      D0.6  ; JB_JZ_JE_COMP_SELECTED_AUX
      OR      D1.5  ; PA_COMP_SELECTED
      OR      D1.7  ; C101_COMP_SELECTED
      ANB
      OUT     F1517  ; SEALENT ROBOT JB SELECT SGNL
; 106
979   LD      D0.0  ; AUTO
      AND     F1514  ; SEALENT ROBOT CYCLE STRT COMM
      OR      D0.1  ; MANUAL
      AND     D0.7  ; DM_BM150_COMP_SELECTED AUX
      OUT     F1516  ; SEALENT ROBOT BM SELECT SGNL
; 107
989   LD      D1410.0  ; SELENT_AUTO_CYCLE_ON
      AND     L1560  ; SEALENT ROBOT CYCLE CMPLT SGNL
      AND     L1561  ; SEALENT ROBOT CYCLE RUNNING SGNL
      SET     D1440.7  ; SEALENT_ROBOT_CYCLE_CMPLT
; 108
997   LD      D1409.6  ; SEALENT_BLANK_COMM
      RST     D1440.7  ; SEALENT_ROBOT_CYCLE_CMPLT
; 110
1003  LD      L1587  ; SEALANT LEVEL LOW
      OUT     T434 K10  ; SEALANT_LEVEL_LOW_TMR
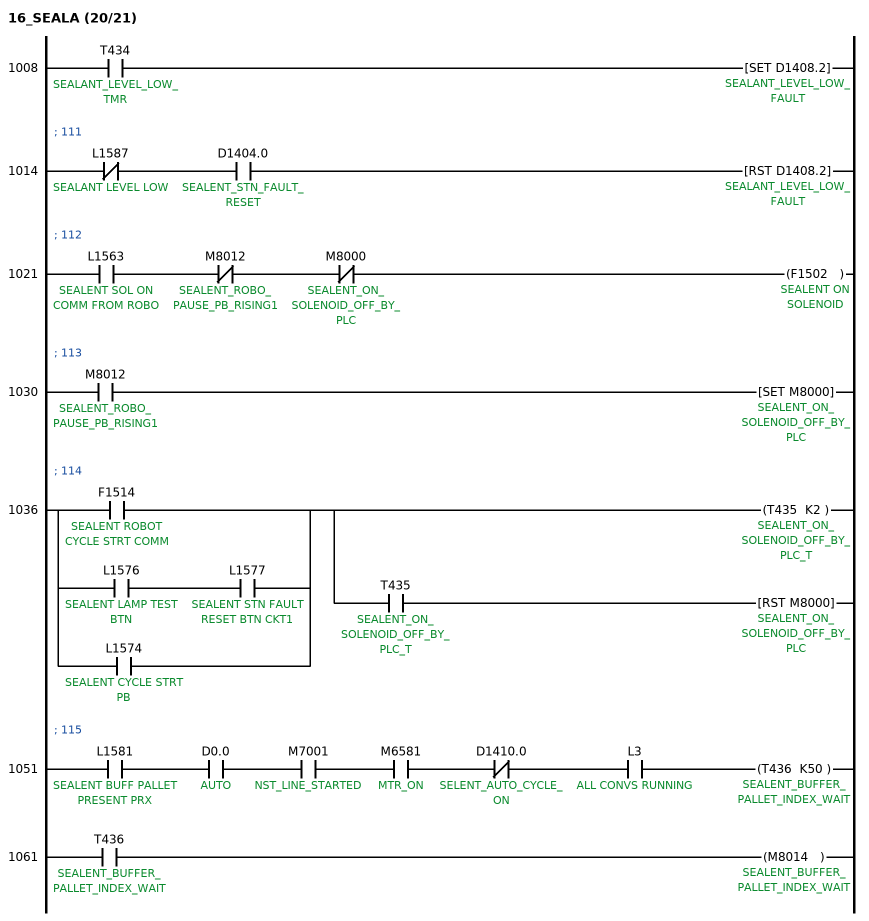
1008  LD      T434  ; SEALANT_LEVEL_LOW_TMR
      SET     D1408.2  ; SEALANT_LEVEL_LOW_FAULT
; 111
1014  LDI     L1587  ; SEALANT LEVEL LOW
      AND     D1404.0  ; SEALENT_STN_FAULT_RESET
      RST     D1408.2  ; SEALANT_LEVEL_LOW_FAULT
; 112
1021  LD      L1563  ; SEALENT SOL ON COMM FROM ROBO
      ANI     M8012  ; SEALENT_ROBO_PAUSE_PB_RISING1
      ANI     M8000  ; SEALENT_ON_SOLENOID_OFF_BY_PLC
      OUT     F1502  ; SEALENT ON SOLENOID
; 113
1030  LD      M8012  ; SEALENT_ROBO_PAUSE_PB_RISING1
      SET     M8000  ; SEALENT_ON_SOLENOID_OFF_BY_PLC
; 114
1036  LD      F1514  ; SEALENT ROBOT CYCLE STRT COMM
      LD      L1576  ; SEALENT LAMP TEST BTN
      AND     L1577  ; SEALENT STN FAULT RESET BTN CKT1
      ORB
      OR      L1574  ; SEALENT CYCLE STRT PB
      OUT     T435 K2  ; SEALENT_ON_SOLENOID_OFF_BY_PLC_T
      AND     T435  ; SEALENT_ON_SOLENOID_OFF_BY_PLC_T
      RST     M8000  ; SEALENT_ON_SOLENOID_OFF_BY_PLC
; 115
1051  LD      L1581  ; SEALENT BUFF PALLET PRESENT PRX
      AND     D0.0  ; AUTO
      AND     M7001  ; NST_LINE_STARTED
      AND     M6581  ; MTR_ON
      ANI     D1410.0  ; SELENT_AUTO_CYCLE_ON
      AND     L3  ; ALL CONVS RUNNING
      OUT     T436 K50  ; SEALENT_BUFFER_PALLET_INDEX_WAIT
1061  LD      T436  ; SEALENT_BUFFER_PALLET_INDEX_WAIT
      OUT     M8014  ; SEALENT_BUFFER_PALLET_INDEX_WAIT
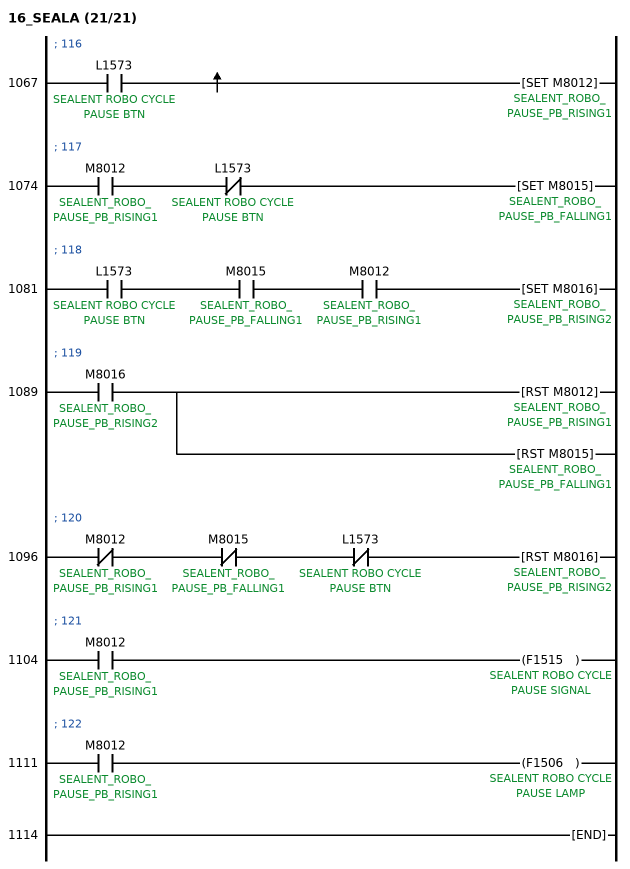
; 116
1067  LD      L1573  ; SEALENT ROBO CYCLE PAUSE BTN
      MEP
      SET     M8012  ; SEALENT_ROBO_PAUSE_PB_RISING1
; 117
1074  LD      M8012  ; SEALENT_ROBO_PAUSE_PB_RISING1
      ANI     L1573  ; SEALENT ROBO CYCLE PAUSE BTN
      SET     M8015  ; SEALENT_ROBO_PAUSE_PB_FALLING1
; 118
1081  LD      L1573  ; SEALENT ROBO CYCLE PAUSE BTN
      AND     M8015  ; SEALENT_ROBO_PAUSE_PB_FALLING1
      AND     M8012  ; SEALENT_ROBO_PAUSE_PB_RISING1
      SET     M8016  ; SEALENT_ROBO_PAUSE_PB_RISING2
; 119
1089  LD      M8016  ; SEALENT_ROBO_PAUSE_PB_RISING2
      RST     M8012  ; SEALENT_ROBO_PAUSE_PB_RISING1
      RST     M8015  ; SEALENT_ROBO_PAUSE_PB_FALLING1
; 120
1096  LDI     M8012  ; SEALENT_ROBO_PAUSE_PB_RISING1
      ANI     M8015  ; SEALENT_ROBO_PAUSE_PB_FALLING1
      ANI     L1573  ; SEALENT ROBO CYCLE PAUSE BTN
      RST     M8016  ; SEALENT_ROBO_PAUSE_PB_RISING2
; 121
1104  LD      M8012  ; SEALENT_ROBO_PAUSE_PB_RISING1
      OUT     F1515  ; SEALENT ROBO CYCLE PAUSE SIGNAL
; 122
1111  LD      M8012  ; SEALENT_ROBO_PAUSE_PB_RISING1
      OUT     F1506  ; SEALENT ROBO CYCLE PAUSE LAMP
1114  END
END_PROGRAM

PROGRAM 17_LOAD  // ST1 CK1
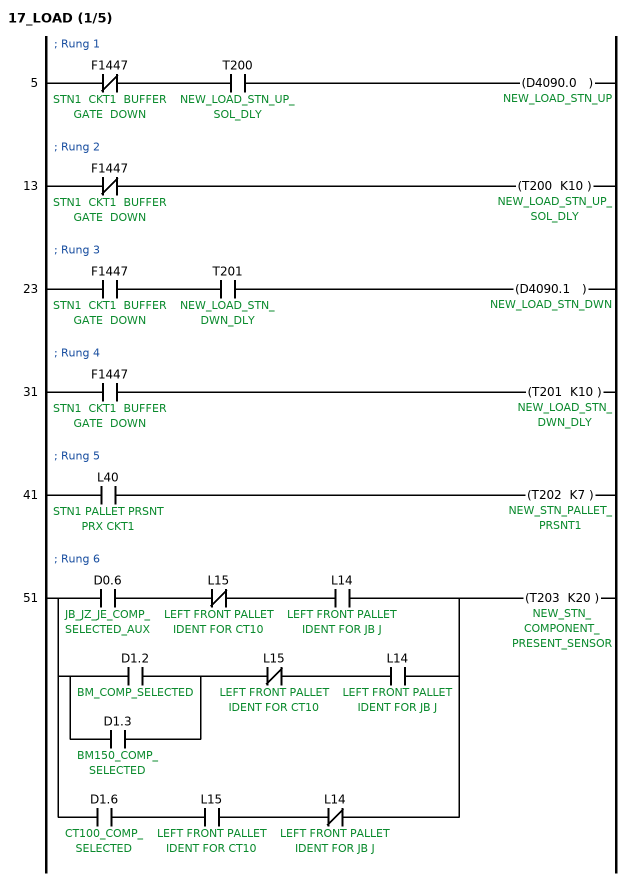
; Rung 1
5     LDI     F1447  ; STN1  CKT1  BUFFER  GATE  DOWN
      AND     T200  ; NEW_LOAD_STN_UP_SOL_DLY
      OUT     D4090.0  ; NEW_LOAD_STN_UP
; Rung 2
13    LDI     F1447  ; STN1  CKT1  BUFFER  GATE  DOWN
      OUT     T200 K10  ; NEW_LOAD_STN_UP_SOL_DLY
; Rung 3
23    LD      F1447  ; STN1  CKT1  BUFFER  GATE  DOWN
      AND     T201  ; NEW_LOAD_STN_DWN_DLY
      OUT     D4090.1  ; NEW_LOAD_STN_DWN
; Rung 4
31    LD      F1447  ; STN1  CKT1  BUFFER  GATE  DOWN
      OUT     T201 K10  ; NEW_LOAD_STN_DWN_DLY
; Rung 5
41    LD      L40  ; STN1 PALLET PRSNT PRX CKT1
      OUT     T202 K7  ; NEW_STN_PALLET_ PRSNT1
; Rung 6
51    LD      D0.6  ; JB_JZ_JE_COMP_SELECTED_AUX
      ANI     L15  ; LEFT FRONT PALLET IDENT FOR CT10
      AND     L14  ; LEFT FRONT PALLET IDENT FOR JB J
      LD      D1.2  ; BM_COMP_SELECTED
      OR      D1.3  ; BM150_COMP_SELECTED
      ANI     L15  ; LEFT FRONT PALLET IDENT FOR CT10
      AND     L14  ; LEFT FRONT PALLET IDENT FOR JB J
      ORB
      LD      D1.6  ; CT100_COMP_SELECTED
      AND     L15  ; LEFT FRONT PALLET IDENT FOR CT10
      ANI     L14  ; LEFT FRONT PALLET IDENT FOR JB J
      ORB
      OUT     T203 K20  ; NEW_STN_COMPONENT_PRESENT_SENSOR
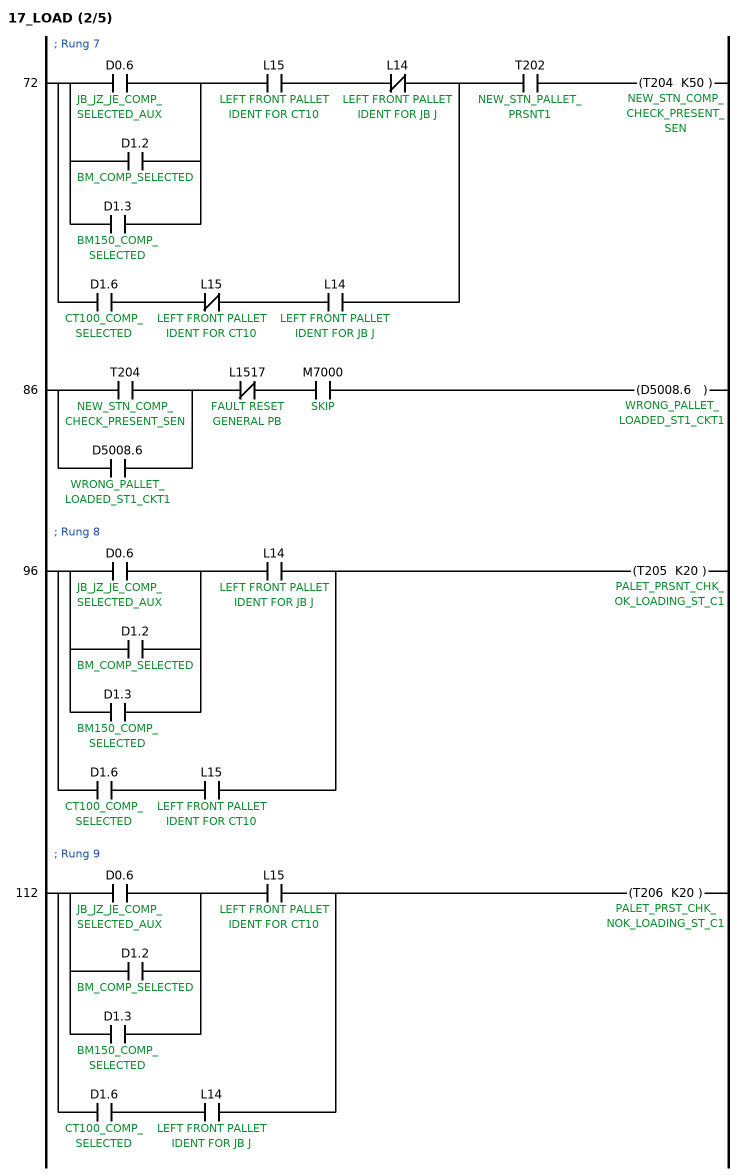
; Rung 7
72    LD      D0.6  ; JB_JZ_JE_COMP_SELECTED_AUX
      OR      D1.2  ; BM_COMP_SELECTED
      OR      D1.3  ; BM150_COMP_SELECTED
      AND     L15  ; LEFT FRONT PALLET IDENT FOR CT10
      ANI     L14  ; LEFT FRONT PALLET IDENT FOR JB J
      LD      D1.6  ; CT100_COMP_SELECTED
      ANI     L15  ; LEFT FRONT PALLET IDENT FOR CT10
      AND     L14  ; LEFT FRONT PALLET IDENT FOR JB J
      ORB
      AND     T202  ; NEW_STN_PALLET_ PRSNT1
      OUT     T204 K50  ; NEW_STN_COMP_CHECK_PRESENT_SEN
86    LD      T204  ; NEW_STN_COMP_CHECK_PRESENT_SEN
      OR      D5008.6  ; WRONG_PALLET_LOADED_ST1_CKT1
      ANI     L1517  ; FAULT RESET GENERAL PB
      AND     M7000  ; SKIP
      OUT     D5008.6  ; WRONG_PALLET_LOADED_ST1_CKT1
; Rung 8
96    LD      D0.6  ; JB_JZ_JE_COMP_SELECTED_AUX
      OR      D1.2  ; BM_COMP_SELECTED
      OR      D1.3  ; BM150_COMP_SELECTED
      AND     L14  ; LEFT FRONT PALLET IDENT FOR JB J
      LD      D1.6  ; CT100_COMP_SELECTED
      AND     L15  ; LEFT FRONT PALLET IDENT FOR CT10
      ORB
      OUT     T205 K20  ; PALET_PRSNT_CHK_OK_LOADING_ST_C1
; Rung 9
112   LD      D0.6  ; JB_JZ_JE_COMP_SELECTED_AUX
      OR      D1.2  ; BM_COMP_SELECTED
      OR      D1.3  ; BM150_COMP_SELECTED
      AND     L15  ; LEFT FRONT PALLET IDENT FOR CT10
      LD      D1.6  ; CT100_COMP_SELECTED
      AND     L14  ; LEFT FRONT PALLET IDENT FOR JB J
      ORB
      OUT     T206 K20  ; PALET_PRST_CHK_NOK_LOADING_ST_C1
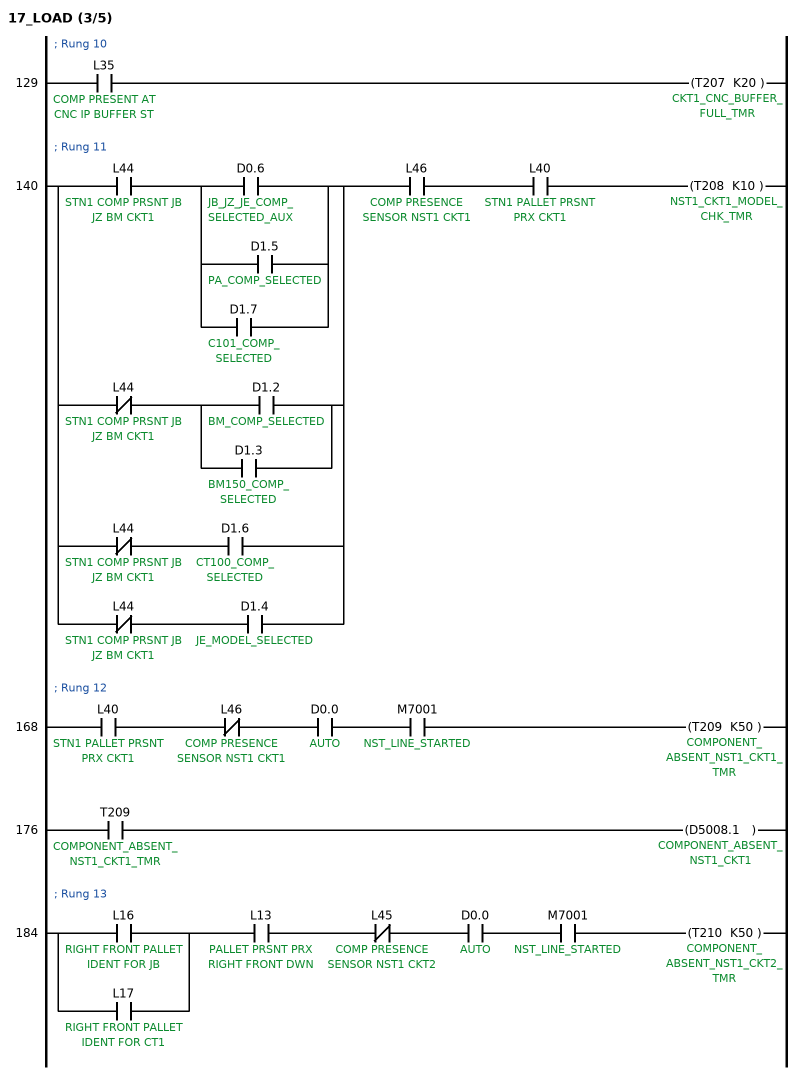
; Rung 10
129   LD      L35  ; COMP PRESENT AT CNC IP BUFFER ST
      OUT     T207 K20  ; CKT1_CNC_BUFFER_FULL_TMR
; Rung 11
140   LD      L44  ; STN1 COMP PRSNT JB JZ BM CKT1
      LD      D0.6  ; JB_JZ_JE_COMP_SELECTED_AUX
      OR      D1.5  ; PA_COMP_SELECTED
      OR      D1.7  ; C101_COMP_SELECTED
      ANB
      LDI     L44  ; STN1 COMP PRSNT JB JZ BM CKT1
      LD      D1.2  ; BM_COMP_SELECTED
      OR      D1.3  ; BM150_COMP_SELECTED
      ANB
      ORB
      LDI     L44  ; STN1 COMP PRSNT JB JZ BM CKT1
      AND     D1.6  ; CT100_COMP_SELECTED
      ORB
      LDI     L44  ; STN1 COMP PRSNT JB JZ BM CKT1
      AND     D1.4  ; JE_MODEL_SELECTED
      ORB
      AND     L46  ; COMP PRESENCE SENSOR NST1 CKT1
      AND     L40  ; STN1 PALLET PRSNT PRX CKT1
      OUT     T208 K10  ; NST1_CKT1_MODEL_CHK_TMR
; Rung 12
168   LD      L40  ; STN1 PALLET PRSNT PRX CKT1
      ANI     L46  ; COMP PRESENCE SENSOR NST1 CKT1
      AND     D0.0  ; AUTO
      AND     M7001  ; NST_LINE_STARTED
      OUT     T209 K50  ; COMPONENT_ABSENT_NST1_CKT1_TMR
176   LD      T209  ; COMPONENT_ABSENT_NST1_CKT1_TMR
      OUT     D5008.1  ; COMPONENT_ABSENT_NST1_CKT1
; Rung 13
184   LD      L16  ; RIGHT FRONT PALLET IDENT FOR JB
      OR      L17  ; RIGHT FRONT PALLET IDENT FOR CT1
      AND     L13  ; PALLET PRSNT PRX RIGHT FRONT DWN
      ANI     L45  ; COMP PRESENCE SENSOR NST1 CKT2
      AND     D0.0  ; AUTO
      AND     M7001  ; NST_LINE_STARTED
      OUT     T210 K50  ; COMPONENT_ABSENT_NST1_CKT2_TMR
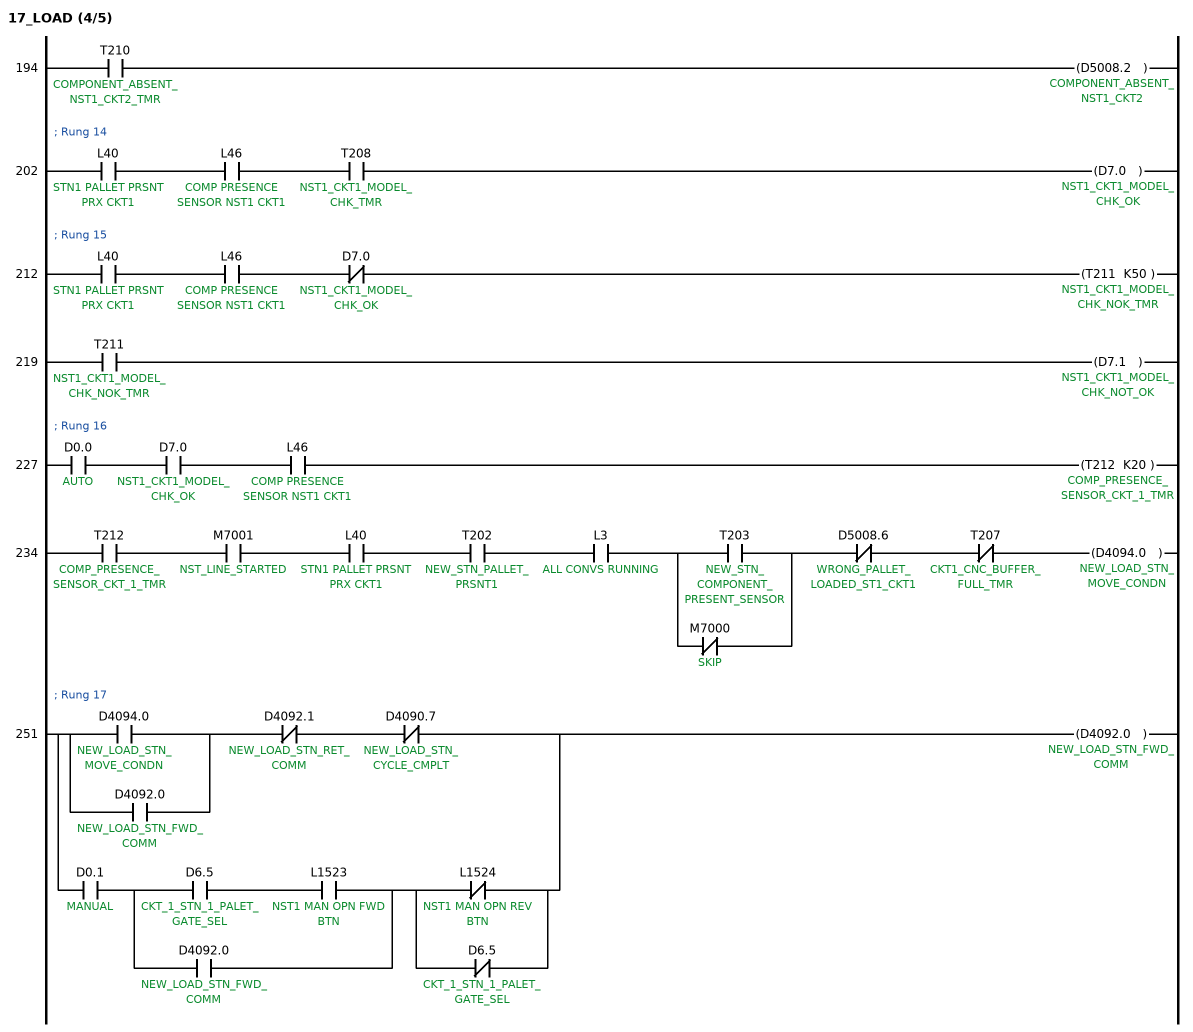
194   LD      T210  ; COMPONENT_ABSENT_NST1_CKT2_TMR
      OUT     D5008.2  ; COMPONENT_ABSENT_NST1_CKT2
; Rung 14
202   LD      L40  ; STN1 PALLET PRSNT PRX CKT1
      AND     L46  ; COMP PRESENCE SENSOR NST1 CKT1
      AND     T208  ; NST1_CKT1_MODEL_CHK_TMR
      OUT     D7.0  ; NST1_CKT1_MODEL_CHK_OK
; Rung 15
212   LD      L40  ; STN1 PALLET PRSNT PRX CKT1
      AND     L46  ; COMP PRESENCE SENSOR NST1 CKT1
      ANI     D7.0  ; NST1_CKT1_MODEL_CHK_OK
      OUT     T211 K50  ; NST1_CKT1_MODEL_CHK_NOK_TMR
219   LD      T211  ; NST1_CKT1_MODEL_CHK_NOK_TMR
      OUT     D7.1  ; NST1_CKT1_MODEL_CHK_NOT_OK
; Rung 16
227   LD      D0.0  ; AUTO
      AND     D7.0  ; NST1_CKT1_MODEL_CHK_OK
      AND     L46  ; COMP PRESENCE SENSOR NST1 CKT1
      OUT     T212 K20  ; COMP_PRESENCE_SENSOR_CKT_1_TMR
234   LD      T212  ; COMP_PRESENCE_SENSOR_CKT_1_TMR
      AND     M7001  ; NST_LINE_STARTED
      AND     L40  ; STN1 PALLET PRSNT PRX CKT1
      AND     T202  ; NEW_STN_PALLET_ PRSNT1
      AND     L3  ; ALL CONVS RUNNING
      LD      T203  ; NEW_STN_COMPONENT_PRESENT_SENSOR
      ORI     M7000  ; SKIP
      ANB
      ANI     D5008.6  ; WRONG_PALLET_LOADED_ST1_CKT1
      ANI     T207  ; CKT1_CNC_BUFFER_FULL_TMR
      OUT     D4094.0  ; NEW_LOAD_STN_MOVE_CONDN
; Rung 17
251   LD      D4094.0  ; NEW_LOAD_STN_MOVE_CONDN
      OR      D4092.0  ; NEW_LOAD_STN_FWD_COMM
      ANI     D4092.1  ; NEW_LOAD_STN_RET_COMM
      ANI     D4090.7  ; NEW_LOAD_STN_CYCLE_CMPLT
      LD      D0.1  ; MANUAL
      LD      D6.5  ; CKT_1_STN_1_PALET_GATE_SEL
      AND     L1523  ; NST1 MAN OPN FWD BTN
      OR      D4092.0  ; NEW_LOAD_STN_FWD_COMM
      ANB
      LDI     L1524  ; NST1 MAN OPN REV BTN
      ORI     D6.5  ; CKT_1_STN_1_PALET_GATE_SEL
      ANB
      ORB
      OUT     D4092.0  ; NEW_LOAD_STN_FWD_COMM
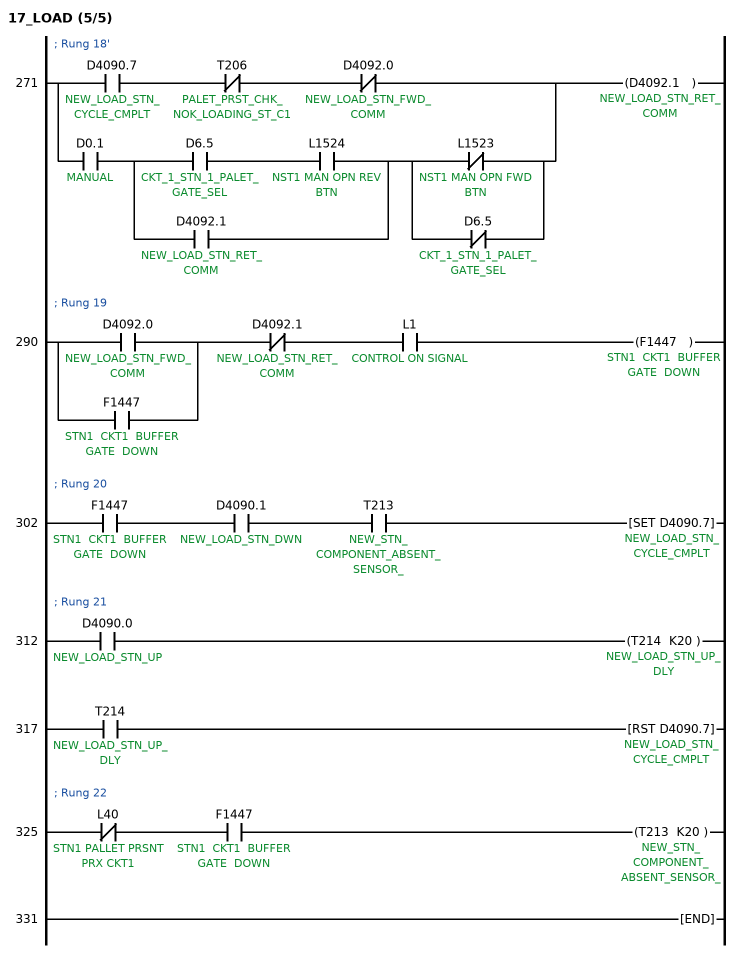
; Rung 18'
271   LD      D4090.7  ; NEW_LOAD_STN_CYCLE_CMPLT
      ANI     T206  ; PALET_PRST_CHK_NOK_LOADING_ST_C1
      ANI     D4092.0  ; NEW_LOAD_STN_FWD_COMM
      LD      D0.1  ; MANUAL
      LD      D6.5  ; CKT_1_STN_1_PALET_GATE_SEL
      AND     L1524  ; NST1 MAN OPN REV BTN
      OR      D4092.1  ; NEW_LOAD_STN_RET_COMM
      ANB
      LDI     L1523  ; NST1 MAN OPN FWD BTN
      ORI     D6.5  ; CKT_1_STN_1_PALET_GATE_SEL
      ANB
      ORB
      OUT     D4092.1  ; NEW_LOAD_STN_RET_COMM
; Rung 19
290   LD      D4092.0  ; NEW_LOAD_STN_FWD_COMM
      OR      F1447  ; STN1  CKT1  BUFFER  GATE  DOWN
      ANI     D4092.1  ; NEW_LOAD_STN_RET_COMM
      AND     L1  ; CONTROL ON SIGNAL
      OUT     F1447  ; STN1  CKT1  BUFFER  GATE  DOWN
; Rung 20
302   LD      F1447  ; STN1  CKT1  BUFFER  GATE  DOWN
      AND     D4090.1  ; NEW_LOAD_STN_DWN
      AND     T213  ; NEW_STN_COMPONENT_ABSENT_SENSOR_
      SET     D4090.7  ; NEW_LOAD_STN_CYCLE_CMPLT
; Rung 21
312   LD      D4090.0  ; NEW_LOAD_STN_UP
      OUT     T214 K20  ; NEW_LOAD_STN_UP_DLY
317   LD      T214  ; NEW_LOAD_STN_UP_DLY
      RST     D4090.7  ; NEW_LOAD_STN_CYCLE_CMPLT
; Rung 22
325   LDI     L40  ; STN1 PALLET PRSNT PRX CKT1
      AND     F1447  ; STN1  CKT1  BUFFER  GATE  DOWN
      OUT     T213 K20  ; NEW_STN_COMPONENT_ABSENT_SENSOR_
331   END
END_PROGRAM

PROGRAM 18_TEST1
